(* PLC project DBISFactory.project, CODESYS CODESYS V3.5 SP10 Patch 5 *)
(* stored: creationDateTime 2019-03-07T13:49:44.3534286, modificationDateTime 2019-03-07T13:47:37.4051931 *)

(* values of BatchJobState: NULL: NULL always expresses that the object has not been initialized yet; WAITING: BatchJob has been initialized and is waiting to be executed; STARTED: BatchJob has been started and is being executed now; PAUSED: BatchJob has been paused during execution; ABORTED: BatchJob has been aborted. This may happen at any time; FINISHED: BatchJob has been finished *)

(* States of a BatchJob Copyright (c) 2019 Manuel Goester, Michael Witt, Klaus Kammerer Institute of Databases and Information Systems, Ulm University, Germany Permission is hereby granted, free of charge, to any person obtaining a copy of this software and associated documentation files (the "Software"), to deal in the Software without restriction, including without limitation the rights to use, copy, modify, merge, publish, distribute, sublicense, and/or sell copies of the Software, and to permit persons to whom the Software is furnished to do so, subject to the following conditions: The above copyright notice and this permission notice shall be included in all copies or substantial portions of the Software. THE SOFTWARE IS PROVIDED "AS IS", WITHOUT WARRANTY OF ANY KIND, EXPRESS OR IMPLIED, INCLUDING BUT NOT LIMITED TO THE WARRANTIES OF MERCHANTABILITY, FITNESS FOR A PARTICULAR PURPOSE AND NONINFRINGEMENT. IN NO EVENT SHALL THE AUTHORS OR COPYRIGHT HOLDERS BE LIABLE FOR ANY CLAIM, DAMAGES OR OTHER LIABILITY, WHETHER IN AN ACTION OF CONTRACT, TORT OR OTHERWISE, ARISING FROM, OUT OF OR IN CONNECTION WITH THE SOFTWARE OR THE USE OR OTHER DEALINGS IN THE SOFTWARE. *)
TYPE BatchJobState : (NULL := 0, WAITING := 1, STARTED := 2, PAUSED := 3, ABORTED := 4, FINISHED := 5);
END_TYPE

(* Execution modes of a BatchJob Copyright (c) 2019 Manuel Goester, Michael Witt, Klaus Kammerer Institute of Databases and Information Systems, Ulm University, Germany Permission is hereby granted, free of charge, to any person obtaining a copy of this software and associated documentation files (the "Software"), to deal in the Software without restriction, including without limitation the rights to use, copy, modify, merge, publish, distribute, sublicense, and/or sell copies of the Software, and to permit persons to whom the Software is furnished to do so, subject to the following conditions: The above copyright notice and this permission notice shall be included in all copies or substantial portions of the Software. THE SOFTWARE IS PROVIDED "AS IS", WITHOUT WARRANTY OF ANY KIND, EXPRESS OR IMPLIED, INCLUDING BUT NOT LIMITED TO THE WARRANTIES OF MERCHANTABILITY, FITNESS FOR A PARTICULAR PURPOSE AND NONINFRINGEMENT. IN NO EVENT SHALL THE AUTHORS OR COPYRIGHT HOLDERS BE LIABLE FOR ANY CLAIM, DAMAGES OR OTHER LIABILITY, WHETHER IN AN ACTION OF CONTRACT, TORT OR OTHERWISE, ARISING FROM, OUT OF OR IN CONNECTION WITH THE SOFTWARE OR THE USE OR OTHER DEALINGS IN THE SOFTWARE. *)
TYPE ExecutionMode : (single := 0, multi := 1, sorting := 2);
END_TYPE

(* A Format defines the execution options of a workpiece Copyright (c) 2019 Manuel Goester, Michael Witt, Klaus Kammerer Institute of Databases and Information Systems, Ulm University, Germany Permission is hereby granted, free of charge, to any person obtaining a copy of this software and associated documentation files (the "Software"), to deal in the Software without restriction, including without limitation the rights to use, copy, modify, merge, publish, distribute, sublicense, and/or sell copies of the Software, and to permit persons to whom the Software is furnished to do so, subject to the following conditions: The above copyright notice and this permission notice shall be included in all copies or substantial portions of the Software. THE SOFTWARE IS PROVIDED "AS IS", WITHOUT WARRANTY OF ANY KIND, EXPRESS OR IMPLIED, INCLUDING BUT NOT LIMITED TO THE WARRANTIES OF MERCHANTABILITY, FITNESS FOR A PARTICULAR PURPOSE AND NONINFRINGEMENT. IN NO EVENT SHALL THE AUTHORS OR COPYRIGHT HOLDERS BE LIABLE FOR ANY CLAIM, DAMAGES OR OTHER LIABILITY, WHETHER IN AN ACTION OF CONTRACT, TORT OR OTHERWISE, ARISING FROM, OUT OF OR IN CONNECTION WITH THE SOFTWARE OR THE USE OR OTHER DEALINGS IN THE SOFTWARE. *)
TYPE Format : STRUCT
  furEnabled : BOOL;
  sawEnabled : BOOL;
  colorCheckEnabled : BOOL;
  ejectEnabled : BOOL;
  furDuration : TIME;
  sawDuration : TIME;
END_STRUCT;
END_TYPE

(* Configured BatchJobs are stored in a BatchJobQueue Copyright (c) 2019 Manuel Goester, Michael Witt, Klaus Kammerer Institute of Databases and Information Systems, Ulm University, Germany Permission is hereby granted, free of charge, to any person obtaining a copy of this software and associated documentation files (the "Software"), to deal in the Software without restriction, including without limitation the rights to use, copy, modify, merge, publish, distribute, sublicense, and/or sell copies of the Software, and to permit persons to whom the Software is furnished to do so, subject to the following conditions: The above copyright notice and this permission notice shall be included in all copies or substantial portions of the Software. THE SOFTWARE IS PROVIDED "AS IS", WITHOUT WARRANTY OF ANY KIND, EXPRESS OR IMPLIED, INCLUDING BUT NOT LIMITED TO THE WARRANTIES OF MERCHANTABILITY, FITNESS FOR A PARTICULAR PURPOSE AND NONINFRINGEMENT. IN NO EVENT SHALL THE AUTHORS OR COPYRIGHT HOLDERS BE LIABLE FOR ANY CLAIM, DAMAGES OR OTHER LIABILITY, WHETHER IN AN ACTION OF CONTRACT, TORT OR OTHERWISE, ARISING FROM, OUT OF OR IN CONNECTION WITH THE SOFTWARE OR THE USE OR OTHER DEALINGS IN THE SOFTWARE. *)
TYPE BatchJobQueue : STRUCT
  batchJobs : ARRAY[1..512] OF BatchJob;  (* batch job queue *)
  nextFreePos : INT := 1;  (* next free place in batchJobs *)
  amountBatchJobs : INT := 0;  (* amount of batch jobs currently being in queue *)
  full : BOOL;  (* true if batchJobs array full *)
END_STRUCT;
END_TYPE

(* Datastructure describing the "real world workpiece" Copyright (c) 2019 Manuel Goester, Michael Witt, Klaus Kammerer Institute of Databases and Information Systems, Ulm University, Germany Permission is hereby granted, free of charge, to any person obtaining a copy of this software and associated documentation files (the "Software"), to deal in the Software without restriction, including without limitation the rights to use, copy, modify, merge, publish, distribute, sublicense, and/or sell copies of the Software, and to permit persons to whom the Software is furnished to do so, subject to the following conditions: The above copyright notice and this permission notice shall be included in all copies or substantial portions of the Software. THE SOFTWARE IS PROVIDED "AS IS", WITHOUT WARRANTY OF ANY KIND, EXPRESS OR IMPLIED, INCLUDING BUT NOT LIMITED TO THE WARRANTIES OF MERCHANTABILITY, FITNESS FOR A PARTICULAR PURPOSE AND NONINFRINGEMENT. IN NO EVENT SHALL THE AUTHORS OR COPYRIGHT HOLDERS BE LIABLE FOR ANY CLAIM, DAMAGES OR OTHER LIABILITY, WHETHER IN AN ACTION OF CONTRACT, TORT OR OTHERWISE, ARISING FROM, OUT OF OR IN CONNECTION WITH THE SOFTWARE OR THE USE OR OTHER DEALINGS IN THE SOFTWARE. *)
TYPE Workpiece : STRUCT
  color : STRING(7);  (* red, blue, white or unknown *)
  linePos : INT;  (* 0 = high rack, 1 = vacuum gripper, 2 = Furnace, 3 = sorting line *)
  sortingLinePos : INT;  (* position in high rack at begin and end of batch job (1,1) (1,2) (1,3) (2,1) (2,2) (2,3) (3,1) (3,2) (3,3) highRackPos: ARRAY [1..2] OF INT; highRackPosEnd: ARRAY [1..2] OF INT; position in sorting line *)
  state : W_State;
  startPos : RackPos;
  endPos : RackPos;
  format : Format;  (* defines which actions will be executed and how long *)
END_STRUCT;
END_TYPE

(* A BatchJob is a task which shall be executed on the production lane. It consists of a set of workpieces, which are executed by the production lane in a certain mode. Copyright (c) 2019 Manuel Goester, Michael Witt, Klaus Kammerer Institute of Databases and Information Systems, Ulm University, Germany Permission is hereby granted, free of charge, to any person obtaining a copy of this software and associated documentation files (the "Software"), to deal in the Software without restriction, including without limitation the rights to use, copy, modify, merge, publish, distribute, sublicense, and/or sell copies of the Software, and to permit persons to whom the Software is furnished to do so, subject to the following conditions: The above copyright notice and this permission notice shall be included in all copies or substantial portions of the Software. THE SOFTWARE IS PROVIDED "AS IS", WITHOUT WARRANTY OF ANY KIND, EXPRESS OR IMPLIED, INCLUDING BUT NOT LIMITED TO THE WARRANTIES OF MERCHANTABILITY, FITNESS FOR A PARTICULAR PURPOSE AND NONINFRINGEMENT. IN NO EVENT SHALL THE AUTHORS OR COPYRIGHT HOLDERS BE LIABLE FOR ANY CLAIM, DAMAGES OR OTHER LIABILITY, WHETHER IN AN ACTION OF CONTRACT, TORT OR OTHERWISE, ARISING FROM, OUT OF OR IN CONNECTION WITH THE SOFTWARE OR THE USE OR OTHER DEALINGS IN THE SOFTWARE. *)
TYPE BatchJob : STRUCT
  batchSize : INT;  (* amount of workpieces in batch job *)
  workpieces : ARRAY[1..9] OF Workpiece;  (* workpieces being processed *)
  nextFreeWPos : INT := 1;  (* next free place in workpieces *)
  nextNotProcessedIdx : INT := 1;  (* index in workpieces of the next workpiece whose production has not started yet *)
  amountFinishedW : INT := 0;  (* states how many workpieces are already finished *)
  mode : ExecutionMode := ExecutionMode.single;  (* type of execution *)
  timeCreated : DT;  (* time when created *)
  timeStarted : DT;  (* time when started *)
  timeFinished : DT;  (* time when finished / aborted *)
  pauseDuration : TIME;  (* states the time how long the batch job was in pause state *)
  duration : TIME;  (* states how long the batch job took *)
  state : BatchJobState := BatchJobState.NULL;  (* state of batch job *)
END_STRUCT;
END_TYPE

(* values of RackPos: UP: there are different values for up position or down position at rack or at conveyor see: HR_FBs/HR_MOVE_TO_POS *)

(* Positions in high rack. Used for HR navigation Copyright (c) 2019 Manuel Goester, Michael Witt, Klaus Kammerer Institute of Databases and Information Systems, Ulm University, Germany Permission is hereby granted, free of charge, to any person obtaining a copy of this software and associated documentation files (the "Software"), to deal in the Software without restriction, including without limitation the rights to use, copy, modify, merge, publish, distribute, sublicense, and/or sell copies of the Software, and to permit persons to whom the Software is furnished to do so, subject to the following conditions: The above copyright notice and this permission notice shall be included in all copies or substantial portions of the Software. THE SOFTWARE IS PROVIDED "AS IS", WITHOUT WARRANTY OF ANY KIND, EXPRESS OR IMPLIED, INCLUDING BUT NOT LIMITED TO THE WARRANTIES OF MERCHANTABILITY, FITNESS FOR A PARTICULAR PURPOSE AND NONINFRINGEMENT. IN NO EVENT SHALL THE AUTHORS OR COPYRIGHT HOLDERS BE LIABLE FOR ANY CLAIM, DAMAGES OR OTHER LIABILITY, WHETHER IN AN ACTION OF CONTRACT, TORT OR OTHERWISE, ARISING FROM, OUT OF OR IN CONNECTION WITH THE SOFTWARE OR THE USE OR OTHER DEALINGS IN THE SOFTWARE. *)
TYPE RackPos : (NULL := 0, RACK_11 := 1, RACK_12 := 2, RACK_13 := 3, RACK_21 := 4, RACK_22 := 5, RACK_23 := 6, RACK_31 := 7, RACK_32 := 8, RACK_33 := 9, CONVEYOR := 10, UP := 11, DOWN := 12);
END_TYPE

(* values of HR_State: NULL: NULL always expresses that the Object has not been initialized yet; AT_DEFAULT_POS: used in single mode; WAIT_FOR_VG_TO_BRING_W: used in multi mode; GET_W: <-- also used in single mode; FINISHED_SORTING_MODE: used in sorting mode *)

(* States of the HR (High Rack) station. Copyright (c) 2019 Manuel Goester, Michael Witt, Klaus Kammerer Institute of Databases and Information Systems, Ulm University, Germany Permission is hereby granted, free of charge, to any person obtaining a copy of this software and associated documentation files (the "Software"), to deal in the Software without restriction, including without limitation the rights to use, copy, modify, merge, publish, distribute, sublicense, and/or sell copies of the Software, and to permit persons to whom the Software is furnished to do so, subject to the following conditions: The above copyright notice and this permission notice shall be included in all copies or substantial portions of the Software. THE SOFTWARE IS PROVIDED "AS IS", WITHOUT WARRANTY OF ANY KIND, EXPRESS OR IMPLIED, INCLUDING BUT NOT LIMITED TO THE WARRANTIES OF MERCHANTABILITY, FITNESS FOR A PARTICULAR PURPOSE AND NONINFRINGEMENT. IN NO EVENT SHALL THE AUTHORS OR COPYRIGHT HOLDERS BE LIABLE FOR ANY CLAIM, DAMAGES OR OTHER LIABILITY, WHETHER IN AN ACTION OF CONTRACT, TORT OR OTHERWISE, ARISING FROM, OUT OF OR IN CONNECTION WITH THE SOFTWARE OR THE USE OR OTHER DEALINGS IN THE SOFTWARE. *)
TYPE HR_State : (NULL := 0, AT_DEFAULT_POS := 1, FINISHED_SINGLE_MODE := 2, AT_CONVEYOR_BOX_FULL := 25, AT_CONVEYOR_BOX_EMPTY := 26, WAIT_FOR_VG_TO_BRING_W := 8, GET_W := 9, GET_BOX := 10, STORE_W := 20, STORE_BOX := 19, WAIT_FOR_VG_TO_PICK_UP_W := 11, READY := 12, FINISHED_SORTING_MODE := 40, SORTING := 41);
END_TYPE

(* values of VG_State: NULL: NULL always expresses that the object has not been initialized yet; FROM_HR_TO_EJECT: used in single mode; TO_FUR_PUT_W: used in multi mode; READY: ready if VG is at default pos or if VG put down a workpiece at HR --> VG is ready for next workpiece; AT_DEFAULT_POS: used in single and multi mode *)

(* States of the VG (Vacuum Gripper) station. Copyright (c) 2019 Manuel Goester, Michael Witt, Klaus Kammerer Institute of Databases and Information Systems, Ulm University, Germany Permission is hereby granted, free of charge, to any person obtaining a copy of this software and associated documentation files (the "Software"), to deal in the Software without restriction, including without limitation the rights to use, copy, modify, merge, publish, distribute, sublicense, and/or sell copies of the Software, and to permit persons to whom the Software is furnished to do so, subject to the following conditions: The above copyright notice and this permission notice shall be included in all copies or substantial portions of the Software. THE SOFTWARE IS PROVIDED "AS IS", WITHOUT WARRANTY OF ANY KIND, EXPRESS OR IMPLIED, INCLUDING BUT NOT LIMITED TO THE WARRANTIES OF MERCHANTABILITY, FITNESS FOR A PARTICULAR PURPOSE AND NONINFRINGEMENT. IN NO EVENT SHALL THE AUTHORS OR COPYRIGHT HOLDERS BE LIABLE FOR ANY CLAIM, DAMAGES OR OTHER LIABILITY, WHETHER IN AN ACTION OF CONTRACT, TORT OR OTHERWISE, ARISING FROM, OUT OF OR IN CONNECTION WITH THE SOFTWARE OR THE USE OR OTHER DEALINGS IN THE SOFTWARE. *)
TYPE VG_State : (NULL := 0, FROM_HR_TO_EJECT := 6, AT_HR := 30, FROM_HR_TO_FUR := 31, AT_SL_OUTPUT_1 := 32, AT_SL_OUTPUT_2 := 33, AT_SL_OUTPUT_3 := 34, WAIT_FOR_SL := 35, AT_EJECT_1 := 36, AT_EJECT_2 := 37, AT_EJECT_3 := 38, TO_SL_OUTPUT_1 := 39, TO_SL_OUTPUT_2 := 40, TO_SL_OUTPUT_3 := 41, FROM_DEFAULT_POS_TO_HR := 43, GET_W_FROM_HR := 44, ABOVE_SL := 56, FROM_SL_TO_HR := 57, DROPPING_W_TO_HR := 59, TO_FUR_PUT_W := 8, TO_FUR_PUT_W_FINISHED := 9, TO_SL_TAKE_W := 10, TO_SL_TAKE_W_FINISHED := 11, TO_HR_PUT_W := 12, TO_HR_PUT_W_FINISHED := 13, TO_HR_TAKE_W := 14, TO_HR_TAKE_W_FINISHED := 15, TO_EJECT := 16, TO_EJECT_FINISHED := 17, TO_SL := 45, READY := 18, AT_DEFAULT_POS := 1, TO_DEFAULT_POS := 5);
END_TYPE

(* values of FUR_State: NULL: TODO : Use these states also in multi mode NULL always expresses that the Object has not been initialized yet; FUR_WAITING_FOR_W: used in single mode FUR is ready to take a new workpiece; FUR_LB_PASSED: Workpiece passed the lightbarrier at waggon; FUR_WAGON_INSIDE: used in single and multi mode Wagon is inside of burner; FUR_BURNED: Furnace is finished with buring the workpiece; FUR_WAGON_OUTSIDE: Wagon is outside of burner; FUR_SUCCER_AT_FUR: used in single mode furnace succer is at furnace; FUR_SUCCER_DOWN_AT_FUR: furnace succer picks up workpiece; FUR_SUCCER_TO_ROTARY_DESK: furnace succer on the way to rotary desk; FUR_SUCCER_AT_ROTARY_DESK: furnace succer at rotary desk; FUR_SUCCER_DOWN_AT_RD: furnace succer puts down workpiece; FUR_SAW_FINISHED: saw has been finished; FUR_SKIP_SAW: saw has been skipped; FUR_W_FINISHED_BACK_TO_DEFAULT: station has finished processing this workpiece *)

(* States of the FUR (Furnace) station. The station is composed of a burner, succer, rotary desk and saw. Copyright (c) 2019 Manuel Goester, Michael Witt, Klaus Kammerer Institute of Databases and Information Systems, Ulm University, Germany Permission is hereby granted, free of charge, to any person obtaining a copy of this software and associated documentation files (the "Software"), to deal in the Software without restriction, including without limitation the rights to use, copy, modify, merge, publish, distribute, sublicense, and/or sell copies of the Software, and to permit persons to whom the Software is furnished to do so, subject to the following conditions: The above copyright notice and this permission notice shall be included in all copies or substantial portions of the Software. THE SOFTWARE IS PROVIDED "AS IS", WITHOUT WARRANTY OF ANY KIND, EXPRESS OR IMPLIED, INCLUDING BUT NOT LIMITED TO THE WARRANTIES OF MERCHANTABILITY, FITNESS FOR A PARTICULAR PURPOSE AND NONINFRINGEMENT. IN NO EVENT SHALL THE AUTHORS OR COPYRIGHT HOLDERS BE LIABLE FOR ANY CLAIM, DAMAGES OR OTHER LIABILITY, WHETHER IN AN ACTION OF CONTRACT, TORT OR OTHERWISE, ARISING FROM, OUT OF OR IN CONNECTION WITH THE SOFTWARE OR THE USE OR OTHER DEALINGS IN THE SOFTWARE. *)
TYPE FUR_State : (NULL := 0, FUR_WAITING_FOR_W := 1, FUR_LB_PASSED := 2, FUR_WAGON_INSIDE := 3, FUR_BURNED := 4, FUR_WAGON_OUTSIDE := 5, FUR_SUCCER_AT_FUR := 6, FUR_SUCCER_DOWN_AT_FUR := 7, FUR_SUCCER_UP_AT_FUR := 8, FUR_SUCCER_TO_ROTARY_DESK := 9, FUR_SUCCER_AT_ROTARY_DESK := 10, FUR_SUCCER_DOWN_AT_RD := 11, FUR_SUCCER_UP_AT_RD := 12, FUR_SAW_FINISHED := 13, FUR_SKIP_SAW := 14, FUR_W_FINISHED_BACK_TO_DEFAULT := 15);
END_TYPE

(* values of SL_State: NULL: NULL always expresses that the object has not been initialized yet; WAITING_FOR_W: SL is ready to process a new workpiece; W_AT_LB: Lightbarrier at SL entry has been passed by a workpiece; THROW_OUT: if no color was detected, the workpiece will be thrown out to trash; W_RECEIVED: SL got a workpiece to process it *)

(* States of the SL (Sorting Line) station. Copyright (c) 2019 Manuel Goester, Michael Witt, Klaus Kammerer Institute of Databases and Information Systems, Ulm University, Germany Permission is hereby granted, free of charge, to any person obtaining a copy of this software and associated documentation files (the "Software"), to deal in the Software without restriction, including without limitation the rights to use, copy, modify, merge, publish, distribute, sublicense, and/or sell copies of the Software, and to permit persons to whom the Software is furnished to do so, subject to the following conditions: The above copyright notice and this permission notice shall be included in all copies or substantial portions of the Software. THE SOFTWARE IS PROVIDED "AS IS", WITHOUT WARRANTY OF ANY KIND, EXPRESS OR IMPLIED, INCLUDING BUT NOT LIMITED TO THE WARRANTIES OF MERCHANTABILITY, FITNESS FOR A PARTICULAR PURPOSE AND NONINFRINGEMENT. IN NO EVENT SHALL THE AUTHORS OR COPYRIGHT HOLDERS BE LIABLE FOR ANY CLAIM, DAMAGES OR OTHER LIABILITY, WHETHER IN AN ACTION OF CONTRACT, TORT OR OTHERWISE, ARISING FROM, OUT OF OR IN CONNECTION WITH THE SOFTWARE OR THE USE OR OTHER DEALINGS IN THE SOFTWARE. *)
TYPE SL_State : (NULL := 0, WAITING_FOR_W := 1, W_AT_LB := 2, W_AT_COLORCHECK := 3, COLORCHECK_FINISHED := 4, W_READY_FOR_SORTING := 5, THROW_OUT := 6, SORTING := 7, WAITING_FOR_VG_TO_PICK_UP_W := 8, EJECT := 9, EJECTED := 10, W_RECEIVED := 11);
END_TYPE

(* values of W_State: NULL: NULL always expresses that the object has not been initialized yet; AT_RACK_11: states at HR; FROM_RACK_TO_CONVEYOR: NOT used; AT_HR: states at VG NOT used; AT_FUR_IN_WAGON: states at FUR; AT_SL_AT_ENTRY_LIGHT_BARRIER: states at SL not used; AT_EJECT_1: states at EJECT point not used *)

(* Workpiece States Copyright (c) 2019 Manuel Goester, Michael Witt, Klaus Kammerer Institute of Databases and Information Systems, Ulm University, Germany Permission is hereby granted, free of charge, to any person obtaining a copy of this software and associated documentation files (the "Software"), to deal in the Software without restriction, including without limitation the rights to use, copy, modify, merge, publish, distribute, sublicense, and/or sell copies of the Software, and to permit persons to whom the Software is furnished to do so, subject to the following conditions: The above copyright notice and this permission notice shall be included in all copies or substantial portions of the Software. THE SOFTWARE IS PROVIDED "AS IS", WITHOUT WARRANTY OF ANY KIND, EXPRESS OR IMPLIED, INCLUDING BUT NOT LIMITED TO THE WARRANTIES OF MERCHANTABILITY, FITNESS FOR A PARTICULAR PURPOSE AND NONINFRINGEMENT. IN NO EVENT SHALL THE AUTHORS OR COPYRIGHT HOLDERS BE LIABLE FOR ANY CLAIM, DAMAGES OR OTHER LIABILITY, WHETHER IN AN ACTION OF CONTRACT, TORT OR OTHERWISE, ARISING FROM, OUT OF OR IN CONNECTION WITH THE SOFTWARE OR THE USE OR OTHER DEALINGS IN THE SOFTWARE. *)
TYPE W_State : (NULL := 0, AT_RACK_11 := 111, AT_RACK_12 := 112, AT_RACK_13 := 113, AT_RACK_21 := 121, AT_RACK_22 := 122, AT_RACK_23 := 123, AT_RACK_31 := 131, AT_RACK_32 := 132, AT_RACK_33 := 133, FROM_RACK_TO_CONVEYOR := 140, AT_CONVEYOR_INSIDE := 141, FROM_CONVEYOR_INSIDE_TO_OUTSIDE := 142, AT_CONVEYOR_OUTSIDE := 143, FROM_CONVEYOR_OUTSIDE_TO_INSIDE := 144, AT_HR := 200, FROM_HR_TO_FUR := 201, FROM_SL_OUTPUT_TO_HR := 202, FROM_SL_OUTPUT_1_TO_HR := 203, FROM_SL_OUTPUT_2_TO_HR := 204, FROM_SL_OUTPUT_3_TO_HR := 205, FROM_SL_TO_EJECT := 206, FROM_SL_OUTPUT_1_TO_EJECT := 207, FROM_SL_OUTPUT_2_TO_EJECT := 208, FROM_SL_OUTPUT_3_TO_EJECT := 209, FROM_FUR_TO_HR := 210, AT_FUR_IN_WAGON := 300, AT_FUR_IN_FUR := 301, AT_FUR_ATTACHED_TO_SUCCER := 302, AT_FUR_ON_ROTARY_DESK := 303, AT_FUR_AT_SAW := 304, AT_FUR_ON_CONVEYOR := 305, AT_SL_AT_ENTRY_LIGHT_BARRIER := 400, AT_SL_AT_COLORCHECK := 401, AT_SL_AT_EXIT_LIGHT_BARRIER := 402, AT_SL_OUTPUT_1 := 403, AT_SL_OUTPUT_2 := 404, AT_SL_OUTPUT_3 := 405, AT_SL_OUTPUT_TRASH := 406, AT_EJECT_1 := 500, AT_EJECT_2 := 501, AT_EJECT_3 := 502);
END_TYPE

(* values of TC_State: NULL: NULL always expresses that the Object has not been initialized yet; W_LOADED: TC has loaded a new workpiece to HR; WAIT_UNTIL_W_FINISHED: TC is waiting until the workpiece has been processed; LOAD_NEXT_W: TC is loading a new workpiece *)

(* States of TC (Task Configurator). Copyright (c) 2019 Manuel Goester, Michael Witt, Klaus Kammerer Institute of Databases and Information Systems, Ulm University, Germany Permission is hereby granted, free of charge, to any person obtaining a copy of this software and associated documentation files (the "Software"), to deal in the Software without restriction, including without limitation the rights to use, copy, modify, merge, publish, distribute, sublicense, and/or sell copies of the Software, and to permit persons to whom the Software is furnished to do so, subject to the following conditions: The above copyright notice and this permission notice shall be included in all copies or substantial portions of the Software. THE SOFTWARE IS PROVIDED "AS IS", WITHOUT WARRANTY OF ANY KIND, EXPRESS OR IMPLIED, INCLUDING BUT NOT LIMITED TO THE WARRANTIES OF MERCHANTABILITY, FITNESS FOR A PARTICULAR PURPOSE AND NONINFRINGEMENT. IN NO EVENT SHALL THE AUTHORS OR COPYRIGHT HOLDERS BE LIABLE FOR ANY CLAIM, DAMAGES OR OTHER LIABILITY, WHETHER IN AN ACTION OF CONTRACT, TORT OR OTHERWISE, ARISING FROM, OUT OF OR IN CONNECTION WITH THE SOFTWARE OR THE USE OR OTHER DEALINGS IN THE SOFTWARE. *)
TYPE TC_State : (NULL := 0, W_LOADED := 1, WAIT_UNTIL_W_FINISHED := 2, LOAD_NEXT_W := 3);
END_TYPE

PROGRAM FUR_SINGLE_MODE
  VAR
    trigger : INT;
    timer : TON;
    sawStopped : BOOL;
    wAtSL : BOOL;
    fin : BOOL;
  END_VAR

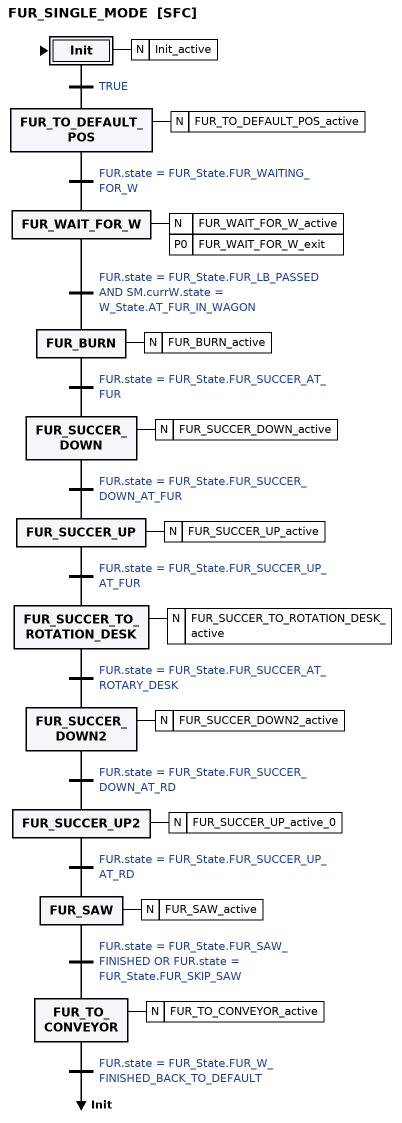
INITIAL_STEP Init:
  Init_active(N);
END_STEP
TRANSITION FROM Init TO FUR_TO_DEFAULT_POS
  := TRUE;
END_TRANSITION
STEP FUR_TO_DEFAULT_POS:
  FUR_TO_DEFAULT_POS_active(N);
END_STEP
TRANSITION FROM FUR_TO_DEFAULT_POS TO FUR_WAIT_FOR_W
  := FUR.state = FUR_State.FUR_WAITING_FOR_W;
END_TRANSITION
STEP FUR_WAIT_FOR_W:
  FUR_WAIT_FOR_W_active(N);
  FUR_WAIT_FOR_W_exit(P0);
END_STEP
TRANSITION FROM FUR_WAIT_FOR_W TO FUR_BURN
  := FUR.state = FUR_State.FUR_LB_PASSED AND SM.currW.state = W_State.AT_FUR_IN_WAGON;
END_TRANSITION
STEP FUR_BURN:
  FUR_BURN_active(N);
END_STEP
TRANSITION FROM FUR_BURN TO FUR_SUCCER_DOWN
  := FUR.state = FUR_State.FUR_SUCCER_AT_FUR;
END_TRANSITION
STEP FUR_SUCCER_DOWN:
  FUR_SUCCER_DOWN_active(N);
END_STEP
TRANSITION FROM FUR_SUCCER_DOWN TO FUR_SUCCER_UP
  := FUR.state = FUR_State.FUR_SUCCER_DOWN_AT_FUR;
END_TRANSITION
STEP FUR_SUCCER_UP:
  FUR_SUCCER_UP_active(N);
END_STEP
TRANSITION FROM FUR_SUCCER_UP TO FUR_SUCCER_TO_ROTATION_DESK
  := FUR.state = FUR_State.FUR_SUCCER_UP_AT_FUR;
END_TRANSITION
STEP FUR_SUCCER_TO_ROTATION_DESK:
  FUR_SUCCER_TO_ROTATION_DESK_active(N);
END_STEP
TRANSITION FROM FUR_SUCCER_TO_ROTATION_DESK TO FUR_SUCCER_DOWN2
  := FUR.state = FUR_State.FUR_SUCCER_AT_ROTARY_DESK;
END_TRANSITION
STEP FUR_SUCCER_DOWN2:
  FUR_SUCCER_DOWN2_active(N);
END_STEP
TRANSITION FROM FUR_SUCCER_DOWN2 TO FUR_SUCCER_UP2
  := FUR.state = FUR_State.FUR_SUCCER_DOWN_AT_RD;
END_TRANSITION
STEP FUR_SUCCER_UP2:
  FUR_SUCCER_UP_active_0(N);
END_STEP
TRANSITION FROM FUR_SUCCER_UP2 TO FUR_SAW
  := FUR.state = FUR_State.FUR_SUCCER_UP_AT_RD;
END_TRANSITION
STEP FUR_SAW:
  FUR_SAW_active(N);
END_STEP
TRANSITION FROM FUR_SAW TO FUR_TO_CONVEYOR
  := FUR.state = FUR_State.FUR_SAW_FINISHED OR FUR.state = FUR_State.FUR_SKIP_SAW;
END_TRANSITION
STEP FUR_TO_CONVEYOR:
  FUR_TO_CONVEYOR_active(N);
END_STEP
TRANSITION FROM FUR_TO_CONVEYOR TO Init
  := FUR.state = FUR_State.FUR_W_FINISHED_BACK_TO_DEFAULT;
END_TRANSITION

ACTION FUR_SUCCER_UP_active_0:
                      (*
Copyright (c) 2019 Manuel Goester, Michael Witt, Klaus Kammerer
Institute of Databases and Information Systems, Ulm University, Germany

Permission is hereby granted, free of charge, to any person obtaining a copy 
of this software and associated documentation files (the "Software"), to deal 
in the Software without restriction, including without limitation the rights 
to use, copy, modify, merge, publish, distribute, sublicense, and/or sell 
copies of the Software, and to permit persons to whom the Software is 
furnished to do so, subject to the following conditions:

The above copyright notice and this permission notice shall be included in 
all copies or substantial portions of the Software.

THE SOFTWARE IS PROVIDED "AS IS", WITHOUT WARRANTY OF ANY KIND, EXPRESS OR 
IMPLIED, INCLUDING BUT NOT LIMITED TO THE WARRANTIES OF MERCHANTABILITY, 
FITNESS FOR A PARTICULAR PURPOSE AND NONINFRINGEMENT. IN NO EVENT SHALL THE 
AUTHORS OR COPYRIGHT HOLDERS BE LIABLE FOR ANY CLAIM, DAMAGES OR OTHER 
LIABILITY, WHETHER IN AN ACTION OF CONTRACT, TORT OR OTHERWISE, ARISING FROM, 
OUT OF OR IN CONNECTION WITH THE SOFTWARE OR THE USE OR OTHER DEALINGS 
IN THE SOFTWARE.
*)
timer(IN:= TRUE, PT := T#200MS);
IF NOT(timer.Q = FALSE AND timer.IN) THEN
	timer(IN:= FALSE);
	FUR.state := FUR_State.FUR_SUCCER_UP_AT_RD;
	SM.currW.state := W_State.AT_FUR_ON_ROTARY_DESK;
END_IF

                    
END_ACTION

ACTION FUR_SUCCER_TO_ROTATION_DESK_active:
                      (*
Copyright (c) 2019 Manuel Goester, Michael Witt, Klaus Kammerer
Institute of Databases and Information Systems, Ulm University, Germany

Permission is hereby granted, free of charge, to any person obtaining a copy 
of this software and associated documentation files (the "Software"), to deal 
in the Software without restriction, including without limitation the rights 
to use, copy, modify, merge, publish, distribute, sublicense, and/or sell 
copies of the Software, and to permit persons to whom the Software is 
furnished to do so, subject to the following conditions:

The above copyright notice and this permission notice shall be included in 
all copies or substantial portions of the Software.

THE SOFTWARE IS PROVIDED "AS IS", WITHOUT WARRANTY OF ANY KIND, EXPRESS OR 
IMPLIED, INCLUDING BUT NOT LIMITED TO THE WARRANTIES OF MERCHANTABILITY, 
FITNESS FOR A PARTICULAR PURPOSE AND NONINFRINGEMENT. IN NO EVENT SHALL THE 
AUTHORS OR COPYRIGHT HOLDERS BE LIABLE FOR ANY CLAIM, DAMAGES OR OTHER 
LIABILITY, WHETHER IN AN ACTION OF CONTRACT, TORT OR OTHERWISE, ARISING FROM, 
OUT OF OR IN CONNECTION WITH THE SOFTWARE OR THE USE OR OTHER DEALINGS 
IN THE SOFTWARE.
*)
IF  NOT(FUR.sSuckerPosRa) THEN
	FUR.mSuckertoRa := TRUE;
	FUR.state := FUR_State.FUR_SUCCER_TO_ROTARY_DESK;
ELSE
	FUR.mSuckertoRa := FALSE;
	FUR.compressor := FALSE;
	FUR.valveLowering := TRUE;
	FUR.state := FUR_State.FUR_SUCCER_AT_ROTARY_DESK;
END_IF
                    
END_ACTION

ACTION FUR_SAW_active:
                      (*
Copyright (c) 2019 Manuel Goester, Michael Witt, Klaus Kammerer
Institute of Databases and Information Systems, Ulm University, Germany

Permission is hereby granted, free of charge, to any person obtaining a copy 
of this software and associated documentation files (the "Software"), to deal 
in the Software without restriction, including without limitation the rights 
to use, copy, modify, merge, publish, distribute, sublicense, and/or sell 
copies of the Software, and to permit persons to whom the Software is 
furnished to do so, subject to the following conditions:

The above copyright notice and this permission notice shall be included in 
all copies or substantial portions of the Software.

THE SOFTWARE IS PROVIDED "AS IS", WITHOUT WARRANTY OF ANY KIND, EXPRESS OR 
IMPLIED, INCLUDING BUT NOT LIMITED TO THE WARRANTIES OF MERCHANTABILITY, 
FITNESS FOR A PARTICULAR PURPOSE AND NONINFRINGEMENT. IN NO EVENT SHALL THE 
AUTHORS OR COPYRIGHT HOLDERS BE LIABLE FOR ANY CLAIM, DAMAGES OR OTHER 
LIABILITY, WHETHER IN AN ACTION OF CONTRACT, TORT OR OTHERWISE, ARISING FROM, 
OUT OF OR IN CONNECTION WITH THE SOFTWARE OR THE USE OR OTHER DEALINGS 
IN THE SOFTWARE.
*)
IF SM.currW.format.sawEnabled THEN
	SM.currW.state := W_State.AT_FUR_AT_SAW;
	IF NOT(FUR.sRaPosSaw) THEN
		FUR.mRaClockwise := TRUE;
	ELSE
		FUR.mRaClockwise := FALSE;
		sawStopped := TRUE;
	END_IF
	
	IF sawStopped THEN
		timer(IN:= TRUE, PT := SM.currW.format.sawDuration);
		FUR.mSaw := TRUE;
		
		IF NOT(timer.Q = FALSE AND timer.IN) THEN
			timer(IN:=FALSE);
			FUR.mSaw := FALSE;
			sawStopped := FALSE;
			FUR.state := FUR_State.FUR_SAW_FINISHED;
		END_IF
	END_IF
ELSE
	// skip saw
	FUR.state := FUR_State.FUR_SKIP_SAW;
END_IF

                    
END_ACTION

ACTION FUR_WAIT_FOR_W_exit:
                      (*
Copyright (c) 2019 Manuel Goester, Michael Witt, Klaus Kammerer
Institute of Databases and Information Systems, Ulm University, Germany

Permission is hereby granted, free of charge, to any person obtaining a copy 
of this software and associated documentation files (the "Software"), to deal 
in the Software without restriction, including without limitation the rights 
to use, copy, modify, merge, publish, distribute, sublicense, and/or sell 
copies of the Software, and to permit persons to whom the Software is 
furnished to do so, subject to the following conditions:

The above copyright notice and this permission notice shall be included in 
all copies or substantial portions of the Software.

THE SOFTWARE IS PROVIDED "AS IS", WITHOUT WARRANTY OF ANY KIND, EXPRESS OR 
IMPLIED, INCLUDING BUT NOT LIMITED TO THE WARRANTIES OF MERCHANTABILITY, 
FITNESS FOR A PARTICULAR PURPOSE AND NONINFRINGEMENT. IN NO EVENT SHALL THE 
AUTHORS OR COPYRIGHT HOLDERS BE LIABLE FOR ANY CLAIM, DAMAGES OR OTHER 
LIABILITY, WHETHER IN AN ACTION OF CONTRACT, TORT OR OTHERWISE, ARISING FROM, 
OUT OF OR IN CONNECTION WITH THE SOFTWARE OR THE USE OR OTHER DEALINGS 
IN THE SOFTWARE.
*)
trigger := 0;
                    
END_ACTION

ACTION Init_active:
                      (*
Copyright (c) 2019 Manuel Goester, Michael Witt, Klaus Kammerer
Institute of Databases and Information Systems, Ulm University, Germany

Permission is hereby granted, free of charge, to any person obtaining a copy 
of this software and associated documentation files (the "Software"), to deal 
in the Software without restriction, including without limitation the rights 
to use, copy, modify, merge, publish, distribute, sublicense, and/or sell 
copies of the Software, and to permit persons to whom the Software is 
furnished to do so, subject to the following conditions:

The above copyright notice and this permission notice shall be included in 
all copies or substantial portions of the Software.

THE SOFTWARE IS PROVIDED "AS IS", WITHOUT WARRANTY OF ANY KIND, EXPRESS OR 
IMPLIED, INCLUDING BUT NOT LIMITED TO THE WARRANTIES OF MERCHANTABILITY, 
FITNESS FOR A PARTICULAR PURPOSE AND NONINFRINGEMENT. IN NO EVENT SHALL THE 
AUTHORS OR COPYRIGHT HOLDERS BE LIABLE FOR ANY CLAIM, DAMAGES OR OTHER 
LIABILITY, WHETHER IN AN ACTION OF CONTRACT, TORT OR OTHERWISE, ARISING FROM, 
OUT OF OR IN CONNECTION WITH THE SOFTWARE OR THE USE OR OTHER DEALINGS 
IN THE SOFTWARE.
*)
FUR.state := -1;
sawStopped := FALSE;
trigger := 0;
                    
END_ACTION

ACTION FUR_SUCCER_DOWN2_active:
                      (*
Copyright (c) 2019 Manuel Goester, Michael Witt, Klaus Kammerer
Institute of Databases and Information Systems, Ulm University, Germany

Permission is hereby granted, free of charge, to any person obtaining a copy 
of this software and associated documentation files (the "Software"), to deal 
in the Software without restriction, including without limitation the rights 
to use, copy, modify, merge, publish, distribute, sublicense, and/or sell 
copies of the Software, and to permit persons to whom the Software is 
furnished to do so, subject to the following conditions:

The above copyright notice and this permission notice shall be included in 
all copies or substantial portions of the Software.

THE SOFTWARE IS PROVIDED "AS IS", WITHOUT WARRANTY OF ANY KIND, EXPRESS OR 
IMPLIED, INCLUDING BUT NOT LIMITED TO THE WARRANTIES OF MERCHANTABILITY, 
FITNESS FOR A PARTICULAR PURPOSE AND NONINFRINGEMENT. IN NO EVENT SHALL THE 
AUTHORS OR COPYRIGHT HOLDERS BE LIABLE FOR ANY CLAIM, DAMAGES OR OTHER 
LIABILITY, WHETHER IN AN ACTION OF CONTRACT, TORT OR OTHERWISE, ARISING FROM, 
OUT OF OR IN CONNECTION WITH THE SOFTWARE OR THE USE OR OTHER DEALINGS 
IN THE SOFTWARE.
*)
IF FUR.sFurnanceSliderOutside THEN
	FUR.compressor := TRUE;
	FUR.valveLowering := TRUE;
	FUR.valveVacuum := FALSE;
	timer(IN:= TRUE, PT := T#1S);
	IF NOT(timer.Q = FALSE AND timer.IN) THEN
		timer(IN:= FALSE);
		FUR.valveLowering := FALSE;
		FUR.state := FUR_State.FUR_SUCCER_DOWN_AT_RD;
	END_IF
END_IF

                    
END_ACTION

ACTION FUR_SUCCER_DOWN_active:
                      (*
Copyright (c) 2019 Manuel Goester, Michael Witt, Klaus Kammerer
Institute of Databases and Information Systems, Ulm University, Germany

Permission is hereby granted, free of charge, to any person obtaining a copy 
of this software and associated documentation files (the "Software"), to deal 
in the Software without restriction, including without limitation the rights 
to use, copy, modify, merge, publish, distribute, sublicense, and/or sell 
copies of the Software, and to permit persons to whom the Software is 
furnished to do so, subject to the following conditions:

The above copyright notice and this permission notice shall be included in 
all copies or substantial portions of the Software.

THE SOFTWARE IS PROVIDED "AS IS", WITHOUT WARRANTY OF ANY KIND, EXPRESS OR 
IMPLIED, INCLUDING BUT NOT LIMITED TO THE WARRANTIES OF MERCHANTABILITY, 
FITNESS FOR A PARTICULAR PURPOSE AND NONINFRINGEMENT. IN NO EVENT SHALL THE 
AUTHORS OR COPYRIGHT HOLDERS BE LIABLE FOR ANY CLAIM, DAMAGES OR OTHER 
LIABILITY, WHETHER IN AN ACTION OF CONTRACT, TORT OR OTHERWISE, ARISING FROM, 
OUT OF OR IN CONNECTION WITH THE SOFTWARE OR THE USE OR OTHER DEALINGS 
IN THE SOFTWARE.
*)
timer(IN:= TRUE, PT := T#2S);
//sauger zum ofen
IF FUR.sFurnanceSliderOutside THEN
	FUR.compressor := TRUE;
	FUR.valveLowering := TRUE;
END_IF

IF NOT(timer.Q = FALSE AND timer.IN) THEN
	// reset timer
	timer(IN:= FALSE);
	// go to next step
	FUR.state := FUR_State.FUR_SUCCER_DOWN_AT_FUR;
END_IF
                    
END_ACTION

ACTION FUR_TO_CONVEYOR_active:
                      (*
Copyright (c) 2019 Manuel Goester, Michael Witt, Klaus Kammerer
Institute of Databases and Information Systems, Ulm University, Germany

Permission is hereby granted, free of charge, to any person obtaining a copy 
of this software and associated documentation files (the "Software"), to deal 
in the Software without restriction, including without limitation the rights 
to use, copy, modify, merge, publish, distribute, sublicense, and/or sell 
copies of the Software, and to permit persons to whom the Software is 
furnished to do so, subject to the following conditions:

The above copyright notice and this permission notice shall be included in 
all copies or substantial portions of the Software.

THE SOFTWARE IS PROVIDED "AS IS", WITHOUT WARRANTY OF ANY KIND, EXPRESS OR 
IMPLIED, INCLUDING BUT NOT LIMITED TO THE WARRANTIES OF MERCHANTABILITY, 
FITNESS FOR A PARTICULAR PURPOSE AND NONINFRINGEMENT. IN NO EVENT SHALL THE 
AUTHORS OR COPYRIGHT HOLDERS BE LIABLE FOR ANY CLAIM, DAMAGES OR OTHER 
LIABILITY, WHETHER IN AN ACTION OF CONTRACT, TORT OR OTHERWISE, ARISING FROM, 
OUT OF OR IN CONNECTION WITH THE SOFTWARE OR THE USE OR OTHER DEALINGS 
IN THE SOFTWARE.
*)
SM.currW.state := W_State.AT_FUR_ON_CONVEYOR;
SL.state := SL_State.W_RECEIVED;
IF NOT(FUR.sRaPosConveyorBelt) THEN
	FUR.mRaClockwise := TRUE;
ELSE
	FUR.mRaClockwise := FALSE;
	FUR.compressor := TRUE;
	FUR.valveSlider := TRUE;
END_IF

IF SL.lbEntry THEN
	FUR.mConveyorBeltForward := TRUE;
ELSE
	FUR.mConveyorBeltForward := FALSE;
	FUR.compressor := FALSE;
	FUR.valveSlider := FALSE;
	FUR.state := FUR_State.FUR_W_FINISHED_BACK_TO_DEFAULT;
END_IF
                    
END_ACTION

ACTION FUR_SUCCER_UP_active:
                      (*
Copyright (c) 2019 Manuel Goester, Michael Witt, Klaus Kammerer
Institute of Databases and Information Systems, Ulm University, Germany

Permission is hereby granted, free of charge, to any person obtaining a copy 
of this software and associated documentation files (the "Software"), to deal 
in the Software without restriction, including without limitation the rights 
to use, copy, modify, merge, publish, distribute, sublicense, and/or sell 
copies of the Software, and to permit persons to whom the Software is 
furnished to do so, subject to the following conditions:

The above copyright notice and this permission notice shall be included in 
all copies or substantial portions of the Software.

THE SOFTWARE IS PROVIDED "AS IS", WITHOUT WARRANTY OF ANY KIND, EXPRESS OR 
IMPLIED, INCLUDING BUT NOT LIMITED TO THE WARRANTIES OF MERCHANTABILITY, 
FITNESS FOR A PARTICULAR PURPOSE AND NONINFRINGEMENT. IN NO EVENT SHALL THE 
AUTHORS OR COPYRIGHT HOLDERS BE LIABLE FOR ANY CLAIM, DAMAGES OR OTHER 
LIABILITY, WHETHER IN AN ACTION OF CONTRACT, TORT OR OTHERWISE, ARISING FROM, 
OUT OF OR IN CONNECTION WITH THE SOFTWARE OR THE USE OR OTHER DEALINGS 
IN THE SOFTWARE.
*)
FUR.valveLowering := FALSE;
FUR.valveVacuum := TRUE; //hier, sonst wird kein vakuum erzeugt
SM.currW.state := W_State.AT_FUR_ATTACHED_TO_SUCCER;
FUR.state := FUR_State.FUR_SUCCER_UP_AT_FUR;
                    
END_ACTION

ACTION FUR_TO_DEFAULT_POS_active:
                      (*
Copyright (c) 2019 Manuel Goester, Michael Witt, Klaus Kammerer
Institute of Databases and Information Systems, Ulm University, Germany

Permission is hereby granted, free of charge, to any person obtaining a copy 
of this software and associated documentation files (the "Software"), to deal 
in the Software without restriction, including without limitation the rights 
to use, copy, modify, merge, publish, distribute, sublicense, and/or sell 
copies of the Software, and to permit persons to whom the Software is 
furnished to do so, subject to the following conditions:

The above copyright notice and this permission notice shall be included in 
all copies or substantial portions of the Software.

THE SOFTWARE IS PROVIDED "AS IS", WITHOUT WARRANTY OF ANY KIND, EXPRESS OR 
IMPLIED, INCLUDING BUT NOT LIMITED TO THE WARRANTIES OF MERCHANTABILITY, 
FITNESS FOR A PARTICULAR PURPOSE AND NONINFRINGEMENT. IN NO EVENT SHALL THE 
AUTHORS OR COPYRIGHT HOLDERS BE LIABLE FOR ANY CLAIM, DAMAGES OR OTHER 
LIABILITY, WHETHER IN AN ACTION OF CONTRACT, TORT OR OTHERWISE, ARISING FROM, 
OUT OF OR IN CONNECTION WITH THE SOFTWARE OR THE USE OR OTHER DEALINGS 
IN THE SOFTWARE.
*)
IF NOT(FUR.sFurnanceSliderOutside) THEN
	FUR.mFurnanceSliderOut := TRUE;
ELSE
	FUR.mFurnanceSliderOut := FALSE;
END_IF

IF NOT(FUR.sSuckerPosRa) THEN
	FUR.mSuckertoRa := TRUE;
ELSE
	FUR.mSuckertoRa := FALSE;
END_IF

IF NOT(FUR.sRaPosSucker) THEN
	FUR.mRaCClockwise := TRUE;
ELSE
	FUR.mRaCClockwise := FALSE;
END_IF

IF FUR.sSuckerPosRa AND FUR.sRaPosSucker AND FUR.sFurnanceSliderOutside THEN
	FUR.state := FUR_WAITING_FOR_W;
END_IF
                    
END_ACTION

ACTION FUR_WAIT_FOR_W_active:
                      (*
Copyright (c) 2019 Manuel Goester, Michael Witt, Klaus Kammerer
Institute of Databases and Information Systems, Ulm University, Germany

Permission is hereby granted, free of charge, to any person obtaining a copy 
of this software and associated documentation files (the "Software"), to deal 
in the Software without restriction, including without limitation the rights 
to use, copy, modify, merge, publish, distribute, sublicense, and/or sell 
copies of the Software, and to permit persons to whom the Software is 
furnished to do so, subject to the following conditions:

The above copyright notice and this permission notice shall be included in 
all copies or substantial portions of the Software.

THE SOFTWARE IS PROVIDED "AS IS", WITHOUT WARRANTY OF ANY KIND, EXPRESS OR 
IMPLIED, INCLUDING BUT NOT LIMITED TO THE WARRANTIES OF MERCHANTABILITY, 
FITNESS FOR A PARTICULAR PURPOSE AND NONINFRINGEMENT. IN NO EVENT SHALL THE 
AUTHORS OR COPYRIGHT HOLDERS BE LIABLE FOR ANY CLAIM, DAMAGES OR OTHER 
LIABILITY, WHETHER IN AN ACTION OF CONTRACT, TORT OR OTHERWISE, ARISING FROM, 
OUT OF OR IN CONNECTION WITH THE SOFTWARE OR THE USE OR OTHER DEALINGS 
IN THE SOFTWARE.
*)
// Workpiece passes the light barrier
IF NOT(FUR.lbFurnance) AND trigger < 2 THEN
	trigger := trigger + 1;
END_IF

// Workpiece passed light barrier
IF FUR.lbFurnance AND trigger >= 2 THEN
	FUR.state := FUR_State.FUR_LB_PASSED;
END_IF


                    
END_ACTION

ACTION FUR_BURN_active:
                      (*
Copyright (c) 2019 Manuel Goester, Michael Witt, Klaus Kammerer
Institute of Databases and Information Systems, Ulm University, Germany

Permission is hereby granted, free of charge, to any person obtaining a copy 
of this software and associated documentation files (the "Software"), to deal 
in the Software without restriction, including without limitation the rights 
to use, copy, modify, merge, publish, distribute, sublicense, and/or sell 
copies of the Software, and to permit persons to whom the Software is 
furnished to do so, subject to the following conditions:

The above copyright notice and this permission notice shall be included in 
all copies or substantial portions of the Software.

THE SOFTWARE IS PROVIDED "AS IS", WITHOUT WARRANTY OF ANY KIND, EXPRESS OR 
IMPLIED, INCLUDING BUT NOT LIMITED TO THE WARRANTIES OF MERCHANTABILITY, 
FITNESS FOR A PARTICULAR PURPOSE AND NONINFRINGEMENT. IN NO EVENT SHALL THE 
AUTHORS OR COPYRIGHT HOLDERS BE LIABLE FOR ANY CLAIM, DAMAGES OR OTHER 
LIABILITY, WHETHER IN AN ACTION OF CONTRACT, TORT OR OTHERWISE, ARISING FROM, 
OUT OF OR IN CONNECTION WITH THE SOFTWARE OR THE USE OR OTHER DEALINGS 
IN THE SOFTWARE.
*)
IF SM.currW.format.furEnabled THEN
	// open door and drive workpiece into furnance 
	IF FUR.state = FUR_State.FUR_LB_PASSED THEN
		FUR.compressor := TRUE;
		FUR.valveFurnanceDoor := TRUE;
		IF FUR.sFurnanceSliderInside = FALSE THEN
			FUR.mFurnanceSliderIn := TRUE;
		ELSE
			FUR.mFurnanceSliderIn := FALSE;
			FUR.state := FUR_State.FUR_WAGON_INSIDE;
		END_IF
	END_IF
	
	// burn
	IF FUR.state = FUR_State.FUR_WAGON_INSIDE THEN
		SM.currW.state := W_State.AT_FUR_IN_FUR;
		timer(IN:= TRUE, PT := SM.currW.format.furDuration);
		FUR.valveFurnanceDoor := FALSE;
		trigger := 0;
		
		// timer finished
		IF NOT(timer.Q = FALSE AND timer.IN) THEN
			timer(IN:= FALSE);
			FUR.compressor := TRUE;
			FUR.valveFurnanceDoor := TRUE;
			FUR.state := FUR_State.FUR_BURNED;
		END_IF
	END_IF
	
	// drive slider out
	IF FUR.state = FUR_State.FUR_BURNED THEN
		SM.currW.state := W_State.AT_FUR_IN_WAGON;
		IF FUR.sFurnanceSliderOutside = FALSE THEN
			FUR.mFurnanceSliderOut := TRUE;
		ELSE
			FUR.mFurnanceSliderOut := FALSE;
			FUR.state := FUR_State.FUR_WAGON_OUTSIDE;
		END_IF
	END_IF
	
	
	// bring succer to furnace
	IF NOT(FUR.sSuckerPosFF) AND (FUR.state = FUR_State.FUR_WAGON_INSIDE OR FUR.state = FUR_State.FUR_BURNED OR FUR.state = FUR_State.FUR_WAGON_OUTSIDE) THEN
		FUR.mSuckertoFurnance := TRUE;
	ELSE
		FUR.mSuckertoFurnance := FALSE;
	END_IF
	
	IF FUR.state = FUR_State.FUR_WAGON_OUTSIDE AND FUR.sSuckerPosFF THEN
		FUR.state := FUR_State.FUR_SUCCER_AT_FUR;
		FUR.mFurnanceSliderOut := FALSE;
		FUR.compressor := FALSE;
		FUR.valveFurnanceDoor := FALSE;
	END_IF
	
ELSE	
	// skip burning
	// bring succer to furnance
	IF NOT(FUR.sSuckerPosFF) THEN
		FUR.mSuckertoFurnance := TRUE;
	ELSE
		FUR.mSuckertoFurnance := FALSE;
		FUR.state := FUR_State.FUR_SUCCER_AT_FUR;
	END_IF
END_IF

                    
END_ACTION
END_PROGRAM

(* Adds a BatchJob to TC.BatchJobQueue Copyright (c) 2019 Manuel Goester, Michael Witt, Klaus Kammerer Institute of Databases and Information Systems, Ulm University, Germany Permission is hereby granted, free of charge, to any person obtaining a copy of this software and associated documentation files (the "Software"), to deal in the Software without restriction, including without limitation the rights to use, copy, modify, merge, publish, distribute, sublicense, and/or sell copies of the Software, and to permit persons to whom the Software is furnished to do so, subject to the following conditions: The above copyright notice and this permission notice shall be included in all copies or substantial portions of the Software. THE SOFTWARE IS PROVIDED "AS IS", WITHOUT WARRANTY OF ANY KIND, EXPRESS OR IMPLIED, INCLUDING BUT NOT LIMITED TO THE WARRANTIES OF MERCHANTABILITY, FITNESS FOR A PARTICULAR PURPOSE AND NONINFRINGEMENT. IN NO EVENT SHALL THE AUTHORS OR COPYRIGHT HOLDERS BE LIABLE FOR ANY CLAIM, DAMAGES OR OTHER LIABILITY, WHETHER IN AN ACTION OF CONTRACT, TORT OR OTHERWISE, ARISING FROM, OUT OF OR IN CONNECTION WITH THE SOFTWARE OR THE USE OR OTHER DEALINGS IN THE SOFTWARE. *)
FUNCTION addBatchJobToQueue : BOOL
  VAR_INPUT
    batchJob : BatchJob;  (* The BatchJob which will be added *)
  END_VAR

                  IF 1 <= TC.batchJobQueue.nextFreePos AND TC.batchJobQueue.nextFreePos <= 20 THEN
	TC.batchJobQueue.batchJobs[TC.batchJobQueue.nextFreePos] := batchJob;
	TC.batchJobQueue.nextFreePos := TC.batchJobQueue.nextFreePos + 1;
	TC.batchJobQueue.amountBatchJobs := TC.batchJobQueue.amountBatchJobs + 1;
	IF TC.batchJobQueue.amountBatchJobs = 20 THEN
		TC.batchJobQueue.full := TRUE;
	ELSE
		TC.batchJobQueue.full := FALSE;
	END_IF
	addBatchJobToQueue := TRUE;
ELSE
	// Batch Job Queue already full
	addBatchJobToQueue := FALSE;	
END_IF
RETURN;
                
END_FUNCTION

(* Constructor for Workpiece Copyright (c) 2019 Manuel Goester, Michael Witt, Klaus Kammerer Institute of Databases and Information Systems, Ulm University, Germany Permission is hereby granted, free of charge, to any person obtaining a copy of this software and associated documentation files (the "Software"), to deal in the Software without restriction, including without limitation the rights to use, copy, modify, merge, publish, distribute, sublicense, and/or sell copies of the Software, and to permit persons to whom the Software is furnished to do so, subject to the following conditions: The above copyright notice and this permission notice shall be included in all copies or substantial portions of the Software. THE SOFTWARE IS PROVIDED "AS IS", WITHOUT WARRANTY OF ANY KIND, EXPRESS OR IMPLIED, INCLUDING BUT NOT LIMITED TO THE WARRANTIES OF MERCHANTABILITY, FITNESS FOR A PARTICULAR PURPOSE AND NONINFRINGEMENT. IN NO EVENT SHALL THE AUTHORS OR COPYRIGHT HOLDERS BE LIABLE FOR ANY CLAIM, DAMAGES OR OTHER LIABILITY, WHETHER IN AN ACTION OF CONTRACT, TORT OR OTHERWISE, ARISING FROM, OUT OF OR IN CONNECTION WITH THE SOFTWARE OR THE USE OR OTHER DEALINGS IN THE SOFTWARE. *)
FUNCTION newWorkpiece : Workpiece
  VAR_INPUT
    color : STRING(7);  (* color of the workpiece: red, blue, white or unknown *)
    state : W_State;  (* state at start: 1ij, i = vertical pos in rack at begin, j = horizontal pos in rack at begin *)
    startPos : RackPos;
    endPos : RackPos;
    format : Format;  (* format for this workpiece *)
  END_VAR

                  newWorkpiece.color := color;
newWorkpiece.format := format;
newWorkpiece.startPos := startPos;
newWorkpiece.endPos := endPos;
newWorkpiece.sortingLinePos := -1;
newWorkpiece.linePos := 0;
newWorkpiece.state := state;
RETURN;
                
END_FUNCTION

PROGRAM SL_SINGLE_MODE
  VAR
    sl_fb : SL_FB;
    step : INT := 1;
    fin : BOOL;
  END_VAR

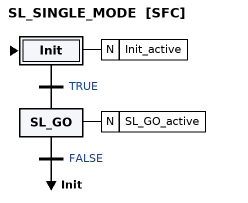
INITIAL_STEP Init:
  Init_active(N);
END_STEP
TRANSITION FROM Init TO SL_GO
  := TRUE;
END_TRANSITION
STEP SL_GO:
  SL_GO_active(N);
END_STEP
TRANSITION FROM SL_GO TO Init
  := FALSE;
END_TRANSITION

ACTION Init_active:
                      (*
Copyright (c) 2019 Manuel Goester, Michael Witt, Klaus Kammerer
Institute of Databases and Information Systems, Ulm University, Germany

Permission is hereby granted, free of charge, to any person obtaining a copy 
of this software and associated documentation files (the "Software"), to deal 
in the Software without restriction, including without limitation the rights 
to use, copy, modify, merge, publish, distribute, sublicense, and/or sell 
copies of the Software, and to permit persons to whom the Software is 
furnished to do so, subject to the following conditions:

The above copyright notice and this permission notice shall be included in 
all copies or substantial portions of the Software.

THE SOFTWARE IS PROVIDED "AS IS", WITHOUT WARRANTY OF ANY KIND, EXPRESS OR 
IMPLIED, INCLUDING BUT NOT LIMITED TO THE WARRANTIES OF MERCHANTABILITY, 
FITNESS FOR A PARTICULAR PURPOSE AND NONINFRINGEMENT. IN NO EVENT SHALL THE 
AUTHORS OR COPYRIGHT HOLDERS BE LIABLE FOR ANY CLAIM, DAMAGES OR OTHER 
LIABILITY, WHETHER IN AN ACTION OF CONTRACT, TORT OR OTHERWISE, ARISING FROM, 
OUT OF OR IN CONNECTION WITH THE SOFTWARE OR THE USE OR OTHER DEALINGS 
IN THE SOFTWARE.
*)
SL.state := SL_State.WAITING_FOR_W;
                    
END_ACTION

ACTION SL_GO_active:
                      (*
Copyright (c) 2019 Manuel Goester, Michael Witt, Klaus Kammerer
Institute of Databases and Information Systems, Ulm University, Germany

Permission is hereby granted, free of charge, to any person obtaining a copy 
of this software and associated documentation files (the "Software"), to deal 
in the Software without restriction, including without limitation the rights 
to use, copy, modify, merge, publish, distribute, sublicense, and/or sell 
copies of the Software, and to permit persons to whom the Software is 
furnished to do so, subject to the following conditions:

The above copyright notice and this permission notice shall be included in 
all copies or substantial portions of the Software.

THE SOFTWARE IS PROVIDED "AS IS", WITHOUT WARRANTY OF ANY KIND, EXPRESS OR 
IMPLIED, INCLUDING BUT NOT LIMITED TO THE WARRANTIES OF MERCHANTABILITY, 
FITNESS FOR A PARTICULAR PURPOSE AND NONINFRINGEMENT. IN NO EVENT SHALL THE 
AUTHORS OR COPYRIGHT HOLDERS BE LIABLE FOR ANY CLAIM, DAMAGES OR OTHER 
LIABILITY, WHETHER IN AN ACTION OF CONTRACT, TORT OR OTHERWISE, ARISING FROM, 
OUT OF OR IN CONNECTION WITH THE SOFTWARE OR THE USE OR OTHER DEALINGS 
IN THE SOFTWARE.
*)
CASE step OF
	1:
		IF SL.state = SL_State.W_RECEIVED THEN
			step := step + 1;
		END_IF
	2:
		IF NOT(fin) THEN
			sl_fb();
			fin := sl_fb.fin;
		ELSE
			// wait for VG to pick up w
			SL.state := SL_State.WAITING_FOR_VG_TO_PICK_UP_W;
			step := step + 1;
		END_IF
	3:
		// reset own pointers
		SL.bIdx := 0;
		SL.wIdx := 0;
		// reset fin
		fin := FALSE;
		step := 1;
		SL.state := SL_State.WAITING_FOR_W;
END_CASE
                    
END_ACTION
END_PROGRAM

(* Adds the workpiece w to the batchJobs queue, if there is a free place in the queue Copyright (c) 2019 Manuel Goester, Michael Witt, Klaus Kammerer Institute of Databases and Information Systems, Ulm University, Germany Permission is hereby granted, free of charge, to any person obtaining a copy of this software and associated documentation files (the "Software"), to deal in the Software without restriction, including without limitation the rights to use, copy, modify, merge, publish, distribute, sublicense, and/or sell copies of the Software, and to permit persons to whom the Software is furnished to do so, subject to the following conditions: The above copyright notice and this permission notice shall be included in all copies or substantial portions of the Software. THE SOFTWARE IS PROVIDED "AS IS", WITHOUT WARRANTY OF ANY KIND, EXPRESS OR IMPLIED, INCLUDING BUT NOT LIMITED TO THE WARRANTIES OF MERCHANTABILITY, FITNESS FOR A PARTICULAR PURPOSE AND NONINFRINGEMENT. IN NO EVENT SHALL THE AUTHORS OR COPYRIGHT HOLDERS BE LIABLE FOR ANY CLAIM, DAMAGES OR OTHER LIABILITY, WHETHER IN AN ACTION OF CONTRACT, TORT OR OTHERWISE, ARISING FROM, OUT OF OR IN CONNECTION WITH THE SOFTWARE OR THE USE OR OTHER DEALINGS IN THE SOFTWARE. *)
FUNCTION addWorkpieceToBatchJob : BOOL
  VAR_INPUT
    batchJob : BatchJob;  (* the batch job *)
    w : workpiece;  (* the workpiece to be added to the batch jobs queue *)
  END_VAR

                  IF batchJob.nextFreeWPos >= 1 AND batchJob.nextFreeWPos <= 9 THEN
	// free place available
	batchJob.workpieces[batchJob.nextFreeWPos] := w;
	batchJob.nextFreeWPos := batchJob.nextFreeWPos + 1;
	batchJob.batchSize := batchJob.batchSize + 1;
	AddWorkpieceToBatchJob := TRUE;
ELSE
	// queue full
	AddWorkpieceToBatchJob := FALSE;
END_IF
RETURN;
                
END_FUNCTION

PROGRAM VG_MULTI_MODE
  VAR
    fin : BOOL;
    step : INT := 1;
    timer : TON;
    sorting_line_pos : INT := -1;
    vg_move_to_pos : VG_MOVE_TO_POS;
    vg_move : VG_MOVE;
  END_VAR

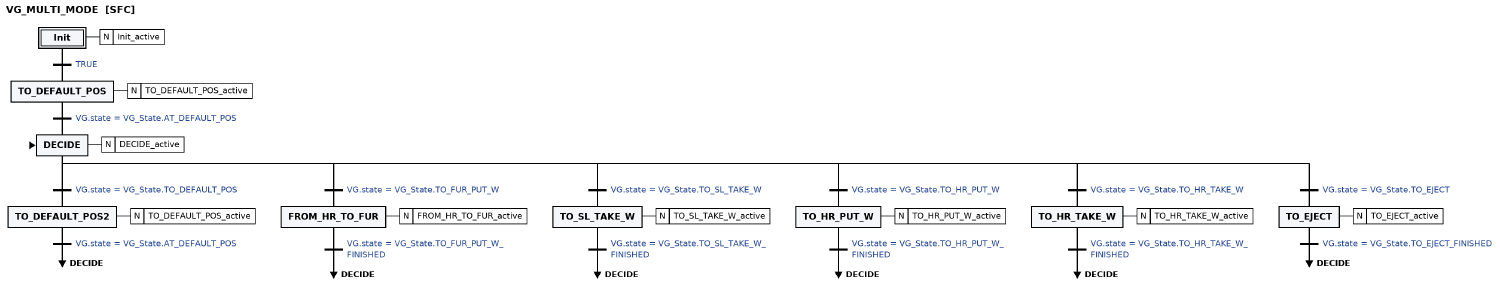
INITIAL_STEP Init:
  Init_active(N);
END_STEP
TRANSITION FROM Init TO TO_DEFAULT_POS
  := TRUE;
END_TRANSITION
STEP TO_DEFAULT_POS:
  TO_DEFAULT_POS_active(N);
END_STEP
TRANSITION FROM TO_DEFAULT_POS TO DECIDE
  := VG.state = VG_State.AT_DEFAULT_POS;
END_TRANSITION
STEP DECIDE:
  DECIDE_active(N);
END_STEP
TRANSITION FROM DECIDE TO TO_DEFAULT_POS2
  := VG.state = VG_State.TO_DEFAULT_POS;
END_TRANSITION
TRANSITION FROM DECIDE TO FROM_HR_TO_FUR
  := VG.state = VG_State.TO_FUR_PUT_W;
END_TRANSITION
TRANSITION FROM DECIDE TO TO_SL_TAKE_W
  := VG.state = VG_State.TO_SL_TAKE_W;
END_TRANSITION
TRANSITION FROM DECIDE TO TO_HR_PUT_W
  := VG.state = VG_State.TO_HR_PUT_W;
END_TRANSITION
TRANSITION FROM DECIDE TO TO_HR_TAKE_W
  := VG.state = VG_State.TO_HR_TAKE_W;
END_TRANSITION
TRANSITION FROM DECIDE TO TO_EJECT
  := VG.state = VG_State.TO_EJECT;
END_TRANSITION
STEP TO_DEFAULT_POS2:
  TO_DEFAULT_POS_active(N);
END_STEP
TRANSITION FROM TO_DEFAULT_POS2 TO DECIDE
  := VG.state = VG_State.AT_DEFAULT_POS;
END_TRANSITION
STEP FROM_HR_TO_FUR:
  FROM_HR_TO_FUR_active(N);
END_STEP
TRANSITION FROM FROM_HR_TO_FUR TO DECIDE
  := VG.state = VG_State.TO_FUR_PUT_W_FINISHED;
END_TRANSITION
STEP TO_SL_TAKE_W:
  TO_SL_TAKE_W_active(N);
END_STEP
TRANSITION FROM TO_SL_TAKE_W TO DECIDE
  := VG.state = VG_State.TO_SL_TAKE_W_FINISHED;
END_TRANSITION
STEP TO_HR_PUT_W:
  TO_HR_PUT_W_active(N);
END_STEP
TRANSITION FROM TO_HR_PUT_W TO DECIDE
  := VG.state = VG_State.TO_HR_PUT_W_FINISHED;
END_TRANSITION
STEP TO_HR_TAKE_W:
  TO_HR_TAKE_W_active(N);
END_STEP
TRANSITION FROM TO_HR_TAKE_W TO DECIDE
  := VG.state = VG_State.TO_HR_TAKE_W_FINISHED;
END_TRANSITION
STEP TO_EJECT:
  TO_EJECT_active(N);
END_STEP
TRANSITION FROM TO_EJECT TO DECIDE
  := VG.state = VG_State.TO_EJECT_FINISHED;
END_TRANSITION

ACTION TO_DEFAULT_POS_active:
                      (*
Copyright (c) 2019 Manuel Goester, Michael Witt, Klaus Kammerer
Institute of Databases and Information Systems, Ulm University, Germany

Permission is hereby granted, free of charge, to any person obtaining a copy 
of this software and associated documentation files (the "Software"), to deal 
in the Software without restriction, including without limitation the rights 
to use, copy, modify, merge, publish, distribute, sublicense, and/or sell 
copies of the Software, and to permit persons to whom the Software is 
furnished to do so, subject to the following conditions:

The above copyright notice and this permission notice shall be included in 
all copies or substantial portions of the Software.

THE SOFTWARE IS PROVIDED "AS IS", WITHOUT WARRANTY OF ANY KIND, EXPRESS OR 
IMPLIED, INCLUDING BUT NOT LIMITED TO THE WARRANTIES OF MERCHANTABILITY, 
FITNESS FOR A PARTICULAR PURPOSE AND NONINFRINGEMENT. IN NO EVENT SHALL THE 
AUTHORS OR COPYRIGHT HOLDERS BE LIABLE FOR ANY CLAIM, DAMAGES OR OTHER 
LIABILITY, WHETHER IN AN ACTION OF CONTRACT, TORT OR OTHERWISE, ARISING FROM, 
OUT OF OR IN CONNECTION WITH THE SOFTWARE OR THE USE OR OTHER DEALINGS 
IN THE SOFTWARE.
*)
// Brings VG to its default pos where sVertical = sHorizontal = sRotation = TRUE
// 1. y-Axis 2. z-Axis 3. rotation
IF NOT(VG.sVertical) THEN
	VG.mVerticalUp := TRUE;
ELSE
	VG.mVerticalUp := FALSE;
	// reset position counter
	VG.cY := 0;
	IF NOT(VG.sHorizontal) THEN
		VG.mHorizontalBackward := TRUE;
	ELSE
		VG.mHorizontalBackward := FALSE;
		// reset position counter
		VG.cX := 0;
		IF NOT(VG.sRotation) THEN
			VG.mRotationClockwise := TRUE;
		ELSE
			VG.mRotationClockwise := FALSE;
			// reset position counter
			VG.cZ := 0;
			
			// wait for 0.5 sec
			timer(IN:= TRUE, PT := T#0.5S);
			IF NOT(timer.Q = FALSE AND timer.IN) THEN
				timer(IN:=FALSE);
				
				// default pos reached
				VG.state := VG_State.AT_DEFAULT_POS;
			END_IF
		END_IF
	END_IF
END_IF
                    
END_ACTION

ACTION DECIDE_active:
                      (*
Copyright (c) 2019 Manuel Goester, Michael Witt, Klaus Kammerer
Institute of Databases and Information Systems, Ulm University, Germany

Permission is hereby granted, free of charge, to any person obtaining a copy 
of this software and associated documentation files (the "Software"), to deal 
in the Software without restriction, including without limitation the rights 
to use, copy, modify, merge, publish, distribute, sublicense, and/or sell 
copies of the Software, and to permit persons to whom the Software is 
furnished to do so, subject to the following conditions:

The above copyright notice and this permission notice shall be included in 
all copies or substantial portions of the Software.

THE SOFTWARE IS PROVIDED "AS IS", WITHOUT WARRANTY OF ANY KIND, EXPRESS OR 
IMPLIED, INCLUDING BUT NOT LIMITED TO THE WARRANTIES OF MERCHANTABILITY, 
FITNESS FOR A PARTICULAR PURPOSE AND NONINFRINGEMENT. IN NO EVENT SHALL THE 
AUTHORS OR COPYRIGHT HOLDERS BE LIABLE FOR ANY CLAIM, DAMAGES OR OTHER 
LIABILITY, WHETHER IN AN ACTION OF CONTRACT, TORT OR OTHERWISE, ARISING FROM, 
OUT OF OR IN CONNECTION WITH THE SOFTWARE OR THE USE OR OTHER DEALINGS 
IN THE SOFTWARE.
*)
IF VG.state = VG_State.AT_HR THEN
	// this can happen if the batch job before was a single mode batch job. Then VG is already AT HR and is not in ready state
	VG.state := VG_State.TO_HR_TAKE_W;
ELSIF VG.state = VG_State.READY AND (HR.state = HR_State.GET_W AND HR.currW.state <> W_State.NULL) THEN
	// go to HR and take w
	VG.state := VG_State.TO_HR_TAKE_W;
ELSIF VG.state = VG_State.READY AND (NOT(SL.lbWhite) OR NOT(SL.lbRed) OR NOT(SL.lbBlue)) AND SL.currW.state <> W_State.NULL AND (NOT(HR.decidedToTakeANewW) OR HR.currW.state = W_State.NULL) THEN
	// go to SL and take w
	// bend VG pointers to workpiece being picked up
	VG.bIdx := SL.bIdx;
	VG.wIdx := SL.wIdx;
	VG.currW := TC.batchJobQueue.batchJobs[VG.bIdx].workpieces[VG.wIdx];
	VG.state := VG_State.TO_SL_TAKE_W;
ELSIF VG.state = VG_State.TO_SL_TAKE_W_FINISHED THEN
	// reset SL pointers
	SL.bIdx := 0;
	SL.wIdx := 0;
	SL.currW := TC.nullW;
	// at SL, w taken, decide if going to EJECT or HR
	IF VG.currW.format.ejectEnabled THEN
		// go to eject point and eject w
		VG.state := VG_State.TO_EJECT;
	ELSE
		// go to HR and put down w
		VG.state := VG_State.TO_HR_PUT_W;
	END_IF
ELSIF VG.state = VG_State.TO_HR_TAKE_W_FINISHED THEN
	// at HR, w taken, decide if going to FUR or EJECT
	IF VG.currW.format.ejectEnabled AND NOT(VG.currW.format.colorCheckEnabled OR VG.currW.format.furEnabled OR VG.currW.format.sawEnabled) THEN
		// go to eject point and eject w
		VG.state := VG_State.TO_EJECT;
	ELSE
		// go to FUR and put down w
		// but only if FUR-succer is at its default pos
		IF FUR.sSuckerPosRa THEN
			VG.state := VG_State.TO_FUR_PUT_W;
		END_IF
	END_IF
ELSIF VG.state = VG_State.TO_EJECT_FINISHED OR VG.state = VG_State.TO_FUR_PUT_W_FINISHED OR  VG.state = VG_State.TO_HR_PUT_W_FINISHED THEN
	// eject or putting w to FUR finished, back to default position for calibrating axes
	// likewise if VG put down w at HR
	VG.state := VG_State.TO_DEFAULT_POS;
ELSIF VG.state = VG_State.AT_DEFAULT_POS THEN
	// state = ready if VG is at default pos or if VG put down a w at HR --> VG is ready for next w
	VG.state := VG_state.READY;
	// reset own pointers
	VG.bIdx := 0;
	VG.wIdx := 0;
	VG.currW := TC.nullW;
END_IF
                    
END_ACTION

ACTION FROM_HR_TO_FUR_active:
                      (*
Copyright (c) 2019 Manuel Goester, Michael Witt, Klaus Kammerer
Institute of Databases and Information Systems, Ulm University, Germany

Permission is hereby granted, free of charge, to any person obtaining a copy 
of this software and associated documentation files (the "Software"), to deal 
in the Software without restriction, including without limitation the rights 
to use, copy, modify, merge, publish, distribute, sublicense, and/or sell 
copies of the Software, and to permit persons to whom the Software is 
furnished to do so, subject to the following conditions:

The above copyright notice and this permission notice shall be included in 
all copies or substantial portions of the Software.

THE SOFTWARE IS PROVIDED "AS IS", WITHOUT WARRANTY OF ANY KIND, EXPRESS OR 
IMPLIED, INCLUDING BUT NOT LIMITED TO THE WARRANTIES OF MERCHANTABILITY, 
FITNESS FOR A PARTICULAR PURPOSE AND NONINFRINGEMENT. IN NO EVENT SHALL THE 
AUTHORS OR COPYRIGHT HOLDERS BE LIABLE FOR ANY CLAIM, DAMAGES OR OTHER 
LIABILITY, WHETHER IN AN ACTION OF CONTRACT, TORT OR OTHERWISE, ARISING FROM, 
OUT OF OR IN CONNECTION WITH THE SOFTWARE OR THE USE OR OTHER DEALINGS 
IN THE SOFTWARE.
*)
CASE step OF
	1:
		// x and z axis: move to FUR
		IF NOT(fin) THEN
			vg_move_to_pos(x := 131, y := 0, z := 137);
			fin := vg_move_to_pos.fin;
		ELSE
			fin := FALSE;
			step := step + 1;
		END_IF
	2:
		// y axis: move to FUR
		IF NOT(fin) THEN
			vg_move_to_pos(x := 131, y := 85, z := 137);
			fin := vg_move_to_pos.fin;
		ELSE
			fin := FALSE;
			step := step + 1;
		END_IF
	3:
		// open ventil to put down w onto waggon
		VG.valve := FALSE;
		step := step + 1;
	4:
		// wait 1 second to get sure w is not succed anymore
		timer(IN:= TRUE, PT:= T#1S);
		IF NOT(timer.Q = FALSE AND timer.IN) THEN
			// reset timer
			timer(IN:= FALSE);
			step := step + 1;
		END_IF
	5:
		// y axis: go up as far as possible
		IF NOT(VG.sVertical) THEN
			VG.mVerticalUp := TRUE;
		ELSE
			VG.mVerticalUp := FALSE;
			// reset y axis counter
			VG.cY := 0;
			// reset step counter
			step := 1;
			// bend FUR-Burner pointers to current workpiece of VG
			FUR.bIdxBurner := VG.bIdx;
			FUR.wIdxBurner := VG.wIdx;
			FUR.currWBurner := TC.batchJobQueue.batchJobs[FUR.bIdxBurner].workpieces[FUR.wIdxBurner];
			// finished
			VG.state := VG_State.TO_FUR_PUT_W_FINISHED;
		END_IF
	6:
	
END_CASE
                    
END_ACTION

ACTION TO_SL_TAKE_W_active:
                      (*
Copyright (c) 2019 Manuel Goester, Michael Witt, Klaus Kammerer
Institute of Databases and Information Systems, Ulm University, Germany

Permission is hereby granted, free of charge, to any person obtaining a copy 
of this software and associated documentation files (the "Software"), to deal 
in the Software without restriction, including without limitation the rights 
to use, copy, modify, merge, publish, distribute, sublicense, and/or sell 
copies of the Software, and to permit persons to whom the Software is 
furnished to do so, subject to the following conditions:

The above copyright notice and this permission notice shall be included in 
all copies or substantial portions of the Software.

THE SOFTWARE IS PROVIDED "AS IS", WITHOUT WARRANTY OF ANY KIND, EXPRESS OR 
IMPLIED, INCLUDING BUT NOT LIMITED TO THE WARRANTIES OF MERCHANTABILITY, 
FITNESS FOR A PARTICULAR PURPOSE AND NONINFRINGEMENT. IN NO EVENT SHALL THE 
AUTHORS OR COPYRIGHT HOLDERS BE LIABLE FOR ANY CLAIM, DAMAGES OR OTHER 
LIABILITY, WHETHER IN AN ACTION OF CONTRACT, TORT OR OTHERWISE, ARISING FROM, 
OUT OF OR IN CONNECTION WITH THE SOFTWARE OR THE USE OR OTHER DEALINGS 
IN THE SOFTWARE.
*)
CASE step OF
	1:
		IF NOT(SL.currW.format.ejectEnabled) THEN
			// set flag to inform HR that VG is taking a w to bring it back to HR
			VG.storeW := TRUE;
			//VG.bIdx := SL.bIdx;
			//VG.wIdx := SL.wIdx;
			//VG.currW := TC.batchJobQueue.batchJobs[VG.bIdx].workpieces[VG.wIdx];
		END_IF
		// select sorting line pos
		IF 	TC.batchJobQueue.batchJobs[SL.bIdx].workpieces[SL.wIdx].format.colorCheckEnabled THEN
			IF TC.batchJobQueue.batchJobs[SL.bIdx].workpieces[SL.wIdx].color = 'white' AND NOT(SL.lbWhite) THEN
				sorting_line_pos := 1;
			ELSIF TC.batchJobQueue.batchJobs[SL.bIdx].workpieces[SL.wIdx].color = 'red' AND NOT(SL.lbRed) THEN
				sorting_line_pos := 2;
			ELSIF TC.batchJobQueue.batchJobs[SL.bIdx].workpieces[SL.wIdx].color = 'blue' AND NOT(SL.lbBlue) THEN
				sorting_line_pos := 3;
			END_IF
		ELSE
			// when color was not checked
			sorting_line_pos := 1;
		END_IF
		step := step + 1;
	2:
		// x and z axis: move to SL
		IF NOT(fin) THEN
			CASE sorting_line_pos OF
				1:
					vg_move_to_pos(x := 58, y := 0, z := 69);
				2:
					vg_move_to_pos(x := 63, y := 0, z := 57);
				3:
					vg_move_to_pos(x := 87, y := 0, z := 47);
			END_CASE
		fin := vg_move_to_pos.fin;
		ELSE
			fin := FALSE;
			step := step + 1;
		END_IF
	3:
		// y axis: move to SL
		IF NOT(fin) THEN
			CASE sorting_line_pos OF
				1:
					vg_move_to_pos(x := 58, y := 125, z := 69);
				2:
					vg_move_to_pos(x := 63, y := 125, z := 57);
				3:
					vg_move_to_pos(x := 87, y := 125, z := 47);
			END_CASE
		fin := vg_move_to_pos.fin;
		ELSE
			fin := FALSE;
			step := step + 1;
		END_IF
	4:
		// succ workpiece at SL
		VG.valve := TRUE;
		timer(IN:= TRUE, PT:= T#2S);
		IF timer.Q = FALSE AND timer.IN THEN
			// go
			VG.compressor := TRUE;
		ELSE
			// stop
			VG.compressor := FALSE;
			// reset timer
			timer(IN:= FALSE);
			step := step + 1;
		END_IF
	5:
		// y axis: go up as far as possible
		IF NOT(VG.sVertical) THEN
			VG.mVerticalUp := TRUE;
		ELSE
			VG.mVerticalUp := FALSE;
			// reset y axis counter
			VG.cY := 0;
			// reset step counter
			step := 1;
			// reset sorting line pos
			sorting_line_pos := -1;
			// finished
			VG.state := VG_State.TO_SL_TAKE_W_FINISHED;
		END_IF
END_CASE
                    
END_ACTION

ACTION TO_HR_PUT_W_active:
                      (*
Copyright (c) 2019 Manuel Goester, Michael Witt, Klaus Kammerer
Institute of Databases and Information Systems, Ulm University, Germany

Permission is hereby granted, free of charge, to any person obtaining a copy 
of this software and associated documentation files (the "Software"), to deal 
in the Software without restriction, including without limitation the rights 
to use, copy, modify, merge, publish, distribute, sublicense, and/or sell 
copies of the Software, and to permit persons to whom the Software is 
furnished to do so, subject to the following conditions:

The above copyright notice and this permission notice shall be included in 
all copies or substantial portions of the Software.

THE SOFTWARE IS PROVIDED "AS IS", WITHOUT WARRANTY OF ANY KIND, EXPRESS OR 
IMPLIED, INCLUDING BUT NOT LIMITED TO THE WARRANTIES OF MERCHANTABILITY, 
FITNESS FOR A PARTICULAR PURPOSE AND NONINFRINGEMENT. IN NO EVENT SHALL THE 
AUTHORS OR COPYRIGHT HOLDERS BE LIABLE FOR ANY CLAIM, DAMAGES OR OTHER 
LIABILITY, WHETHER IN AN ACTION OF CONTRACT, TORT OR OTHERWISE, ARISING FROM, 
OUT OF OR IN CONNECTION WITH THE SOFTWARE OR THE USE OR OTHER DEALINGS 
IN THE SOFTWARE.
*)
CASE step OF
	1:
		// x and z axis: move to HR
		IF NOT(fin) THEN
			vg_move_to_pos(x := 27, y := 0, z := 206);
			fin := vg_move_to_pos.fin;
		ELSE
			fin := FALSE;
			step := step + 1;
		END_IF
	2:
		// box without workpiece arrived, wait 0.5 sec to be sure
		IF NOT(HR.lbOut) AND HR.state = HR_State.WAIT_FOR_VG_TO_BRING_W THEN
			timer(IN:= TRUE, PT:= T#0.5S);
			IF NOT(timer.Q = FALSE AND timer.IN) THEN
				timer(IN:= FALSE);
				step := step + 1;
			END_IF
		END_IF
	3:
		// y axis: move down at HR
		IF NOT(fin) THEN
			vg_move_to_pos(x:=27, y:=40, z:=206);
			fin := vg_move_to_pos.fin;
		ELSE
			fin := FALSE;
			step := step + 1;
		END_IF
	4:
		// open ventil
		VG.valve := FALSE;
		step := step + 1;
	5:
		timer(IN:= TRUE, PT:= T#1S);
		IF NOT(timer.Q = FALSE AND timer.IN) THEN
			// reset timer
			timer(IN:= FALSE);
			// go to next step
			step := step + 1;
		END_IF
	6:
		// y axis: go up as far as possible
		IF NOT(VG.sVertical) THEN
			VG.mVerticalUp := TRUE;
		ELSE
			VG.mVerticalUp := FALSE;
			// reset y axis counter
			VG.cY := 0;
			// reset step counter
			step := 1;
			// finished
			VG.state := VG_State.TO_HR_PUT_W_FINISHED;
		END_IF
END_CASE
                    
END_ACTION

ACTION TO_HR_TAKE_W_active:
                      (*
Copyright (c) 2019 Manuel Goester, Michael Witt, Klaus Kammerer
Institute of Databases and Information Systems, Ulm University, Germany

Permission is hereby granted, free of charge, to any person obtaining a copy 
of this software and associated documentation files (the "Software"), to deal 
in the Software without restriction, including without limitation the rights 
to use, copy, modify, merge, publish, distribute, sublicense, and/or sell 
copies of the Software, and to permit persons to whom the Software is 
furnished to do so, subject to the following conditions:

The above copyright notice and this permission notice shall be included in 
all copies or substantial portions of the Software.

THE SOFTWARE IS PROVIDED "AS IS", WITHOUT WARRANTY OF ANY KIND, EXPRESS OR 
IMPLIED, INCLUDING BUT NOT LIMITED TO THE WARRANTIES OF MERCHANTABILITY, 
FITNESS FOR A PARTICULAR PURPOSE AND NONINFRINGEMENT. IN NO EVENT SHALL THE 
AUTHORS OR COPYRIGHT HOLDERS BE LIABLE FOR ANY CLAIM, DAMAGES OR OTHER 
LIABILITY, WHETHER IN AN ACTION OF CONTRACT, TORT OR OTHERWISE, ARISING FROM, 
OUT OF OR IN CONNECTION WITH THE SOFTWARE OR THE USE OR OTHER DEALINGS 
IN THE SOFTWARE.
*)
CASE step OF
	1:
		// x and z axis: move to HR
		IF NOT(fin) THEN
			vg_move_to_pos(x := 27, y := 0, z := 206);
			fin := vg_move_to_pos.fin;
		ELSE
			fin := FALSE;
			step := step + 1;
		END_IF
	2:
		IF NOT(HR.lbOut) THEN
			// box with workpiece arrived, wait 0.5 sec to be sure
			timer(IN:= TRUE, PT:= T#0.5S);
			IF NOT(timer.Q = FALSE AND timer.IN) THEN
				timer(IN:= FALSE);
				step := step + 1;
			END_IF		
		END_IF
	3:
		// y axis: move down at HR
		IF NOT(fin) THEN
			vg_move_to_pos(x:=27, y:=40, z:=206);
			fin := vg_move_to_pos.fin;
		ELSE
			fin := FALSE;
			step := step + 1;
		END_IF
	4:
		// succ w at HR
		VG.valve := TRUE;
		timer(IN:= TRUE, PT:= T#2S);
		IF timer.Q = FALSE AND timer.IN THEN
			// go
			VG.compressor := TRUE;
		ELSE
			// stop
			VG.compressor := FALSE;
			// reset timer
			timer(IN:= FALSE);
			step := step + 1;
		END_IF	
	5:
		// y axis: go up as far as possible
		IF NOT(VG.sVertical) THEN
			VG.mVerticalUp := TRUE;
		ELSE
			VG.mVerticalUp := FALSE;
			// reset y axis counter
			VG.cY := 0;
			// reset step counter
			step := 1;
			// finished
			VG.state := VG_State.TO_HR_TAKE_W_FINISHED;
		END_IF
END_CASE
                    
END_ACTION

ACTION TO_EJECT_active:
                      (*
Copyright (c) 2019 Manuel Goester, Michael Witt, Klaus Kammerer
Institute of Databases and Information Systems, Ulm University, Germany

Permission is hereby granted, free of charge, to any person obtaining a copy 
of this software and associated documentation files (the "Software"), to deal 
in the Software without restriction, including without limitation the rights 
to use, copy, modify, merge, publish, distribute, sublicense, and/or sell 
copies of the Software, and to permit persons to whom the Software is 
furnished to do so, subject to the following conditions:

The above copyright notice and this permission notice shall be included in 
all copies or substantial portions of the Software.

THE SOFTWARE IS PROVIDED "AS IS", WITHOUT WARRANTY OF ANY KIND, EXPRESS OR 
IMPLIED, INCLUDING BUT NOT LIMITED TO THE WARRANTIES OF MERCHANTABILITY, 
FITNESS FOR A PARTICULAR PURPOSE AND NONINFRINGEMENT. IN NO EVENT SHALL THE 
AUTHORS OR COPYRIGHT HOLDERS BE LIABLE FOR ANY CLAIM, DAMAGES OR OTHER 
LIABILITY, WHETHER IN AN ACTION OF CONTRACT, TORT OR OTHERWISE, ARISING FROM, 
OUT OF OR IN CONNECTION WITH THE SOFTWARE OR THE USE OR OTHER DEALINGS 
IN THE SOFTWARE.
*)
CASE step OF
	1:
		// x and z axis: move to EJECT
		IF NOT(fin) THEN
			IF VG.currW.color = 'white' THEN
				// go to eject point 1
				vg_move_to_pos(x := 25, y := 0, z := 2);
			ELSIF VG.currW.color = 'red' THEN
				// go to eject point 2
				vg_move_to_pos(x := 30, y := 0, z := 15);
			ELSIF VG.currW.color = 'blue' THEN
				// go to eject point 3
				vg_move_to_pos(x := 49, y := 0, z := 23);
			ELSE
				// if color 'unknown' then eject to white eject point
				// go to eject point 1
				vg_move_to_pos(x := 25, y := 0, z := 2);
			END_IF
			fin := vg_move_to_pos.fin;
		ELSE
			fin := FALSE;
			step := step + 1;
		END_IF
	2:
		// x and z axis: move to EJECT
		IF NOT(fin) THEN
			IF VG.currW.color = 'white' THEN
				// go to eject point 1
				vg_move_to_pos(x := 25, y := 133, z := 2);
			ELSIF VG.currW.color = 'red' THEN
				// go to eject point 2
				vg_move_to_pos(x := 30, y := 133, z := 15);
			ELSIF VG.currW.color = 'blue' THEN
				// go to eject point 3
				vg_move_to_pos(x := 49, y := 133, z := 23);
			ELSE
				// if color 'unknown' then eject to white eject point
				// go to eject point 1
				vg_move_to_pos(x := 25, y := 133, z := 2);
			END_IF
			fin := vg_move_to_pos.fin;
		ELSE
			fin := FALSE;
			step := step + 1;
		END_IF
	3:
		// open valve to drop w
		VG.valve := FALSE;
		timer(IN:= TRUE, PT:= T#1S);
		IF NOT(timer.Q = FALSE AND timer.IN) THEN
			// reset timer
			timer(IN:= FALSE);
			// reset step counter
			step := 1;
			// finished
			VG.state := VG_State.TO_EJECT_FINISHED;
		END_IF
END_CASE
                    
END_ACTION

ACTION Init_active:
                      (*
Copyright (c) 2019 Manuel Goester, Michael Witt, Klaus Kammerer
Institute of Databases and Information Systems, Ulm University, Germany

Permission is hereby granted, free of charge, to any person obtaining a copy 
of this software and associated documentation files (the "Software"), to deal 
in the Software without restriction, including without limitation the rights 
to use, copy, modify, merge, publish, distribute, sublicense, and/or sell 
copies of the Software, and to permit persons to whom the Software is 
furnished to do so, subject to the following conditions:

The above copyright notice and this permission notice shall be included in 
all copies or substantial portions of the Software.

THE SOFTWARE IS PROVIDED "AS IS", WITHOUT WARRANTY OF ANY KIND, EXPRESS OR 
IMPLIED, INCLUDING BUT NOT LIMITED TO THE WARRANTIES OF MERCHANTABILITY, 
FITNESS FOR A PARTICULAR PURPOSE AND NONINFRINGEMENT. IN NO EVENT SHALL THE 
AUTHORS OR COPYRIGHT HOLDERS BE LIABLE FOR ANY CLAIM, DAMAGES OR OTHER 
LIABILITY, WHETHER IN AN ACTION OF CONTRACT, TORT OR OTHERWISE, ARISING FROM, 
OUT OF OR IN CONNECTION WITH THE SOFTWARE OR THE USE OR OTHER DEALINGS 
IN THE SOFTWARE.
*)
step := 1;
                    
END_ACTION
END_PROGRAM

PROGRAM TC_POU
  VAR
    started : BOOL;  (* true if user pressed start button *)
    batch_job_available : BOOL := FALSE;  (* true if theres a batch job waiting to be executed *)
    fin : BOOL;
    Copyright : INT;
  END_VAR

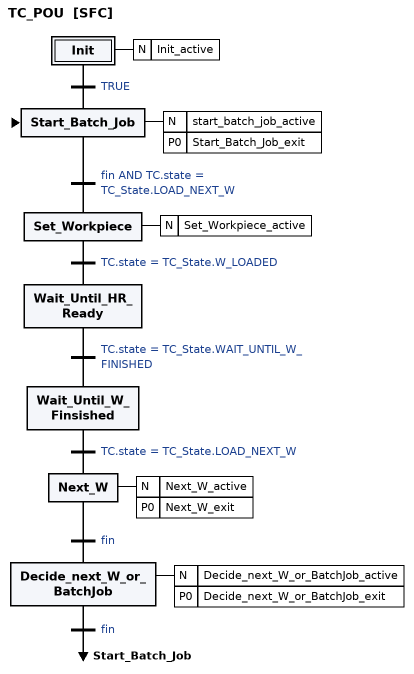
INITIAL_STEP Init:
  Init_active(N);
END_STEP
TRANSITION FROM Init TO Start_Batch_Job
  := TRUE;
END_TRANSITION
STEP Start_Batch_Job:
  start_batch_job_active(N);
  Start_Batch_Job_exit(P0);
END_STEP
TRANSITION FROM Start_Batch_Job TO Set_Workpiece
  := fin AND TC.state = TC_State.LOAD_NEXT_W;
END_TRANSITION
STEP Set_Workpiece:
  Set_Workpiece_active(N);
END_STEP
TRANSITION FROM Set_Workpiece TO Wait_Until_HR_Ready
  := TC.state = TC_State.W_LOADED;
END_TRANSITION
STEP Wait_Until_HR_Ready:
END_STEP
TRANSITION FROM Wait_Until_HR_Ready TO Wait_Until_W_Finsished
  := TC.state = TC_State.WAIT_UNTIL_W_FINISHED;
END_TRANSITION
STEP Wait_Until_W_Finsished:
END_STEP
TRANSITION FROM Wait_Until_W_Finsished TO Next_W
  := TC.state = TC_State.LOAD_NEXT_W;
END_TRANSITION
STEP Next_W:
  Next_W_active(N);
  Next_W_exit(P0);
END_STEP
TRANSITION FROM Next_W TO Decide_next_W_or_BatchJob
  := fin;
END_TRANSITION
STEP Decide_next_W_or_BatchJob:
  Decide_next_W_or_BatchJob_active(N);
  Decide_next_W_or_BatchJob_exit(P0);
END_STEP
TRANSITION FROM Decide_next_W_or_BatchJob TO Start_Batch_Job
  := fin;
END_TRANSITION

ACTION Decide_next_W_or_BatchJob_active:
                      (*
Copyright (c) 2019 Manuel Goester, Michael Witt, Klaus Kammerer
Institute of Databases and Information Systems, Ulm University, Germany

Permission is hereby granted, free of charge, to any person obtaining a copy 
of this software and associated documentation files (the "Software"), to deal 
in the Software without restriction, including without limitation the rights 
to use, copy, modify, merge, publish, distribute, sublicense, and/or sell 
copies of the Software, and to permit persons to whom the Software is 
furnished to do so, subject to the following conditions:

The above copyright notice and this permission notice shall be included in 
all copies or substantial portions of the Software.

THE SOFTWARE IS PROVIDED "AS IS", WITHOUT WARRANTY OF ANY KIND, EXPRESS OR 
IMPLIED, INCLUDING BUT NOT LIMITED TO THE WARRANTIES OF MERCHANTABILITY, 
FITNESS FOR A PARTICULAR PURPOSE AND NONINFRINGEMENT. IN NO EVENT SHALL THE 
AUTHORS OR COPYRIGHT HOLDERS BE LIABLE FOR ANY CLAIM, DAMAGES OR OTHER 
LIABILITY, WHETHER IN AN ACTION OF CONTRACT, TORT OR OTHERWISE, ARISING FROM, 
OUT OF OR IN CONNECTION WITH THE SOFTWARE OR THE USE OR OTHER DEALINGS 
IN THE SOFTWARE.
*)
IF NOT(fin) THEN
	IF TC.batchJobQueue.batchJobs[TC.currBatchJobIdx].nextNotProcessedIdx > TC.batchJobQueue.batchJobs[TC.currBatchJobIdx].batchSize THEN
		IF SM.currW.state = 0 AND HR.bIdx = 0 AND VG.bIdx = 0 AND FUR.bIdxBurner = 0 AND FUR.bIdxSuccer = 0 AND FUR.bIdxSaw = 0 AND SL.bIdx = 0 THEN
			// there is no new workpiece in current BatchJob and all maschines finished processing --> BatchJob finished
			TC.batchJobQueue.batchJobs[TC.currBatchJobIdx].state := BatchJobState.FINISHED;
			// delete finished BatchJob
			TC.batchJobQueue.batchJobs[TC.currBatchJobIdx] := TC.nullB;
			// update counter of BatchJobs in queue
			TC.batchJobQueue.amountBatchJobs := TC.batchJobQueue.amountBatchJobs - 1;
			// start next batch job if there is one
			TC.currBatchJobIdx := TC.currBatchJobIdx + 1;
			IF TC.currBatchJobIdx > 20 THEN
				TC.currBatchJobIdx := 1;
			END_IF
			fin := TRUE;
		END_IF
	ELSE
		// batch job not finished --> execute steps for next workpiece
		fin := TRUE;
	END_IF
END_IF
                    
END_ACTION

ACTION Set_Workpiece_active:
                      (*
Copyright (c) 2019 Manuel Goester, Michael Witt, Klaus Kammerer
Institute of Databases and Information Systems, Ulm University, Germany

Permission is hereby granted, free of charge, to any person obtaining a copy 
of this software and associated documentation files (the "Software"), to deal 
in the Software without restriction, including without limitation the rights 
to use, copy, modify, merge, publish, distribute, sublicense, and/or sell 
copies of the Software, and to permit persons to whom the Software is 
furnished to do so, subject to the following conditions:

The above copyright notice and this permission notice shall be included in 
all copies or substantial portions of the Software.

THE SOFTWARE IS PROVIDED "AS IS", WITHOUT WARRANTY OF ANY KIND, EXPRESS OR 
IMPLIED, INCLUDING BUT NOT LIMITED TO THE WARRANTIES OF MERCHANTABILITY, 
FITNESS FOR A PARTICULAR PURPOSE AND NONINFRINGEMENT. IN NO EVENT SHALL THE 
AUTHORS OR COPYRIGHT HOLDERS BE LIABLE FOR ANY CLAIM, DAMAGES OR OTHER 
LIABILITY, WHETHER IN AN ACTION OF CONTRACT, TORT OR OTHERWISE, ARISING FROM, 
OUT OF OR IN CONNECTION WITH THE SOFTWARE OR THE USE OR OTHER DEALINGS 
IN THE SOFTWARE.
*)
IF TC.batchJobQueue.batchJobs[TC.currBatchJobIdx].state = BatchJobState.NULL THEN
	// no batchjob available
	// wait until new batchjob is loaded
ELSIF TC.batchJobQueue.batchJobs[TC.currBatchJobIdx].mode = ExecutionMode.single THEN
	SM.currW := TC.batchJobQueue.batchJobs[TC.currBatchJobIdx].workpieces[TC.batchJobQueue.batchJobs[TC.currBatchJobIdx].nextNotProcessedIdx];
	IF SM.currW.format.ejectEnabled AND NOT(SM.currW.format.furEnabled) AND NOT(SM.currW.format.sawEnabled) AND NOT(SM.currW.format.colorCheckEnabled) THEN
		// dont set SL flags because workpiece will directly be ejected HR -> VG -> EJECT
		SL.bIdx := 0;
		SL.wIdx := 0;
	ELSE
		// set SL pointers
		SL.bIdx := TC.currBatchJobIdx;
		SL.wIdx := TC.batchJobQueue.batchJobs[TC.currBatchJobIdx].nextNotProcessedIdx;
	END_IF
	TC.state := TC_State.W_LOADED;
ELSIF TC.batchJobQueue.batchJobs[TC.currBatchJobIdx].mode = ExecutionMode.multi AND (HR.state = HR_State.READY OR HR.state = HR_State.FINISHED_SINGLE_MODE OR HR.state = HR_State.SORTING) THEN
	// new w loaded in TC, load it to HR.currW
	Hr.bIdx := TC.currBatchJobIdx;
	Hr.wIdx := TC.batchJobQueue.batchJobs[TC.currBatchJobIdx].nextNotProcessedIdx;
	HR.currW := TC.batchJobQueue.batchJobs[Hr.bIdx].workpieces[Hr.wIdx];
	TC.state := TC_State.W_LOADED;
ELSIF TC.batchJobQueue.batchJobs[TC.currBatchJobIdx].mode = ExecutionMode.sorting THEN
	TC.state := TC_State.W_LOADED;
END_IF
                    
END_ACTION

ACTION start_batch_job_active:
                      (*
Copyright (c) 2019 Manuel Goester, Michael Witt, Klaus Kammerer
Institute of Databases and Information Systems, Ulm University, Germany

Permission is hereby granted, free of charge, to any person obtaining a copy 
of this software and associated documentation files (the "Software"), to deal 
in the Software without restriction, including without limitation the rights 
to use, copy, modify, merge, publish, distribute, sublicense, and/or sell 
copies of the Software, and to permit persons to whom the Software is 
furnished to do so, subject to the following conditions:

The above copyright notice and this permission notice shall be included in 
all copies or substantial portions of the Software.

THE SOFTWARE IS PROVIDED "AS IS", WITHOUT WARRANTY OF ANY KIND, EXPRESS OR 
IMPLIED, INCLUDING BUT NOT LIMITED TO THE WARRANTIES OF MERCHANTABILITY, 
FITNESS FOR A PARTICULAR PURPOSE AND NONINFRINGEMENT. IN NO EVENT SHALL THE 
AUTHORS OR COPYRIGHT HOLDERS BE LIABLE FOR ANY CLAIM, DAMAGES OR OTHER 
LIABILITY, WHETHER IN AN ACTION OF CONTRACT, TORT OR OTHERWISE, ARISING FROM, 
OUT OF OR IN CONNECTION WITH THE SOFTWARE OR THE USE OR OTHER DEALINGS 
IN THE SOFTWARE.
*)
IF started THEN
	IF NOT(fin) THEN
		IF TC.batchJobQueue.batchJobs[TC.currBatchJobIdx].state <> BatchJobState.NULL THEN
			IF TC.batchJobQueue.batchJobs[TC.currBatchJobIdx].mode = ExecutionMode.single THEN
				// start single mode
				TC.mode_active := ExecutionMode.single;
				TC.batchJobQueue.batchJobs[TC.currBatchJobIdx].state := BatchJobState.STARTED;
				fin := TRUE;
			ELSIF TC.batchJobQueue.batchJobs[TC.currBatchJobIdx].mode = ExecutionMode.multi THEN
				// start multi mode
				TC.mode_active := ExecutionMode.multi;
				TC.batchJobQueue.batchJobs[TC.currBatchJobIdx].state := BatchJobState.STARTED;
				fin := TRUE;
			ELSIF TC.batchJobQueue.batchJobs[TC.currBatchJobIdx].mode = ExecutionMode.sorting THEN
				// start sorting mode
				TC.mode_active := ExecutionMode.sorting;
				TC.batchJobQueue.batchJobs[TC.currBatchJobIdx].state := BatchJobState.STARTED;
				fin := TRUE;
			END_IF
		ELSE
			// currently no BatchJob available
			// reset HR pointers, cause they may still set
			HR.bIdx := 0;
			HR.wIdx := 0;
			HR.currW := TC.nullW;
		END_IF
	END_IF
END_IF
                    
END_ACTION

ACTION Init_active:
                      (*
Copyright (c) 2019 Manuel Goester, Michael Witt, Klaus Kammerer
Institute of Databases and Information Systems, Ulm University, Germany

Permission is hereby granted, free of charge, to any person obtaining a copy 
of this software and associated documentation files (the "Software"), to deal 
in the Software without restriction, including without limitation the rights 
to use, copy, modify, merge, publish, distribute, sublicense, and/or sell 
copies of the Software, and to permit persons to whom the Software is 
furnished to do so, subject to the following conditions:

The above copyright notice and this permission notice shall be included in 
all copies or substantial portions of the Software.

THE SOFTWARE IS PROVIDED "AS IS", WITHOUT WARRANTY OF ANY KIND, EXPRESS OR 
IMPLIED, INCLUDING BUT NOT LIMITED TO THE WARRANTIES OF MERCHANTABILITY, 
FITNESS FOR A PARTICULAR PURPOSE AND NONINFRINGEMENT. IN NO EVENT SHALL THE 
AUTHORS OR COPYRIGHT HOLDERS BE LIABLE FOR ANY CLAIM, DAMAGES OR OTHER 
LIABILITY, WHETHER IN AN ACTION OF CONTRACT, TORT OR OTHERWISE, ARISING FROM, 
OUT OF OR IN CONNECTION WITH THE SOFTWARE OR THE USE OR OTHER DEALINGS 
IN THE SOFTWARE.
*)
TC.state := TC_State.NULL;
                    
END_ACTION

ACTION Next_W_active:
                      (*
Copyright (c) 2019 Manuel Goester, Michael Witt, Klaus Kammerer
Institute of Databases and Information Systems, Ulm University, Germany

Permission is hereby granted, free of charge, to any person obtaining a copy 
of this software and associated documentation files (the "Software"), to deal 
in the Software without restriction, including without limitation the rights 
to use, copy, modify, merge, publish, distribute, sublicense, and/or sell 
copies of the Software, and to permit persons to whom the Software is 
furnished to do so, subject to the following conditions:

The above copyright notice and this permission notice shall be included in 
all copies or substantial portions of the Software.

THE SOFTWARE IS PROVIDED "AS IS", WITHOUT WARRANTY OF ANY KIND, EXPRESS OR 
IMPLIED, INCLUDING BUT NOT LIMITED TO THE WARRANTIES OF MERCHANTABILITY, 
FITNESS FOR A PARTICULAR PURPOSE AND NONINFRINGEMENT. IN NO EVENT SHALL THE 
AUTHORS OR COPYRIGHT HOLDERS BE LIABLE FOR ANY CLAIM, DAMAGES OR OTHER 
LIABILITY, WHETHER IN AN ACTION OF CONTRACT, TORT OR OTHERWISE, ARISING FROM, 
OUT OF OR IN CONNECTION WITH THE SOFTWARE OR THE USE OR OTHER DEALINGS 
IN THE SOFTWARE.
*)
// updates the current workpiece pointer to the next workpiece
IF NOT(fin) THEN
	IF NOT(TC.batchJobQueue.batchJobs[TC.currBatchJobIdx].mode = ExecutionMode.sorting) THEN
		TC.batchJobQueue.batchJobs[TC.currBatchJobIdx].nextNotProcessedIdx := TC.batchJobQueue.batchJobs[TC.currBatchJobIdx].nextNotProcessedIdx + 1;
	ELSE
		// in sorting mode always two workpieces are processed simultaniously, so increment by 2
		TC.batchJobQueue.batchJobs[TC.currBatchJobIdx].nextNotProcessedIdx := TC.batchJobQueue.batchJobs[TC.currBatchJobIdx].nextNotProcessedIdx + 2;
	END_IF
	fin := TRUE;
END_IF
                    
END_ACTION

ACTION Next_W_exit:
                      (*
Copyright (c) 2019 Manuel Goester, Michael Witt, Klaus Kammerer
Institute of Databases and Information Systems, Ulm University, Germany

Permission is hereby granted, free of charge, to any person obtaining a copy 
of this software and associated documentation files (the "Software"), to deal 
in the Software without restriction, including without limitation the rights 
to use, copy, modify, merge, publish, distribute, sublicense, and/or sell 
copies of the Software, and to permit persons to whom the Software is 
furnished to do so, subject to the following conditions:

The above copyright notice and this permission notice shall be included in 
all copies or substantial portions of the Software.

THE SOFTWARE IS PROVIDED "AS IS", WITHOUT WARRANTY OF ANY KIND, EXPRESS OR 
IMPLIED, INCLUDING BUT NOT LIMITED TO THE WARRANTIES OF MERCHANTABILITY, 
FITNESS FOR A PARTICULAR PURPOSE AND NONINFRINGEMENT. IN NO EVENT SHALL THE 
AUTHORS OR COPYRIGHT HOLDERS BE LIABLE FOR ANY CLAIM, DAMAGES OR OTHER 
LIABILITY, WHETHER IN AN ACTION OF CONTRACT, TORT OR OTHERWISE, ARISING FROM, 
OUT OF OR IN CONNECTION WITH THE SOFTWARE OR THE USE OR OTHER DEALINGS 
IN THE SOFTWARE.
*)
fin := FALSE;
                    
END_ACTION

ACTION Decide_next_W_or_BatchJob_exit:
                      (*
Copyright (c) 2019 Manuel Goester, Michael Witt, Klaus Kammerer
Institute of Databases and Information Systems, Ulm University, Germany

Permission is hereby granted, free of charge, to any person obtaining a copy 
of this software and associated documentation files (the "Software"), to deal 
in the Software without restriction, including without limitation the rights 
to use, copy, modify, merge, publish, distribute, sublicense, and/or sell 
copies of the Software, and to permit persons to whom the Software is 
furnished to do so, subject to the following conditions:

The above copyright notice and this permission notice shall be included in 
all copies or substantial portions of the Software.

THE SOFTWARE IS PROVIDED "AS IS", WITHOUT WARRANTY OF ANY KIND, EXPRESS OR 
IMPLIED, INCLUDING BUT NOT LIMITED TO THE WARRANTIES OF MERCHANTABILITY, 
FITNESS FOR A PARTICULAR PURPOSE AND NONINFRINGEMENT. IN NO EVENT SHALL THE 
AUTHORS OR COPYRIGHT HOLDERS BE LIABLE FOR ANY CLAIM, DAMAGES OR OTHER 
LIABILITY, WHETHER IN AN ACTION OF CONTRACT, TORT OR OTHERWISE, ARISING FROM, 
OUT OF OR IN CONNECTION WITH THE SOFTWARE OR THE USE OR OTHER DEALINGS 
IN THE SOFTWARE.
*)
fin := FALSE;
                    
END_ACTION

ACTION Start_Batch_Job_exit:
                      (*
Copyright (c) 2019 Manuel Goester, Michael Witt, Klaus Kammerer
Institute of Databases and Information Systems, Ulm University, Germany

Permission is hereby granted, free of charge, to any person obtaining a copy 
of this software and associated documentation files (the "Software"), to deal 
in the Software without restriction, including without limitation the rights 
to use, copy, modify, merge, publish, distribute, sublicense, and/or sell 
copies of the Software, and to permit persons to whom the Software is 
furnished to do so, subject to the following conditions:

The above copyright notice and this permission notice shall be included in 
all copies or substantial portions of the Software.

THE SOFTWARE IS PROVIDED "AS IS", WITHOUT WARRANTY OF ANY KIND, EXPRESS OR 
IMPLIED, INCLUDING BUT NOT LIMITED TO THE WARRANTIES OF MERCHANTABILITY, 
FITNESS FOR A PARTICULAR PURPOSE AND NONINFRINGEMENT. IN NO EVENT SHALL THE 
AUTHORS OR COPYRIGHT HOLDERS BE LIABLE FOR ANY CLAIM, DAMAGES OR OTHER 
LIABILITY, WHETHER IN AN ACTION OF CONTRACT, TORT OR OTHERWISE, ARISING FROM, 
OUT OF OR IN CONNECTION WITH THE SOFTWARE OR THE USE OR OTHER DEALINGS 
IN THE SOFTWARE.
*)
fin := FALSE;
                    
END_ACTION
END_PROGRAM

(* Moves HR in x and y axis Copyright (c) 2019 Manuel Goester, Michael Witt, Klaus Kammerer Institute of Databases and Information Systems, Ulm University, Germany Permission is hereby granted, free of charge, to any person obtaining a copy of this software and associated documentation files (the "Software"), to deal in the Software without restriction, including without limitation the rights to use, copy, modify, merge, publish, distribute, sublicense, and/or sell copies of the Software, and to permit persons to whom the Software is furnished to do so, subject to the following conditions: The above copyright notice and this permission notice shall be included in all copies or substantial portions of the Software. THE SOFTWARE IS PROVIDED "AS IS", WITHOUT WARRANTY OF ANY KIND, EXPRESS OR IMPLIED, INCLUDING BUT NOT LIMITED TO THE WARRANTIES OF MERCHANTABILITY, FITNESS FOR A PARTICULAR PURPOSE AND NONINFRINGEMENT. IN NO EVENT SHALL THE AUTHORS OR COPYRIGHT HOLDERS BE LIABLE FOR ANY CLAIM, DAMAGES OR OTHER LIABILITY, WHETHER IN AN ACTION OF CONTRACT, TORT OR OTHERWISE, ARISING FROM, OUT OF OR IN CONNECTION WITH THE SOFTWARE OR THE USE OR OTHER DEALINGS IN THE SOFTWARE. *)
FUNCTION_BLOCK HR_MOVE
  VAR_INPUT
    x : INT;  (* distance HR will go right (negative value) or left (positive value) *)
    y : INT;  (* distance HR will go up (negative value) or down (positive value) *)
  END_VAR
  VAR
    xFin : BOOL := FALSE;  (* finish flags *)
    yFin : BOOL := FALSE;
    fin : BOOL := FALSE;
    xAlreadyCounted : BOOL := FALSE;  (* true, if an impulse coming from the motor has been already counted *)
    yAlreadyCounted : BOOL := FALSE;
    cX : INT := 0;  (* counters for x and y axis *)
    cY : INT := 0;
  END_VAR

                  fin := FALSE;

// X AXIS
IF x < 0 THEN
	// drive right
	IF cX = x THEN
		// if counter reached demanded position, we're done
		HR.mHorizontalRight := FALSE;
		HR.mHorizontalLeft := FALSE;
		xFin := TRUE;
	ELSE
		xFin := FALSE;
		IF cX > x THEN
			HR.mHorizontalRight := TRUE;
			IF HR.encHorizontal AND NOT(xAlreadyCounted) THEN
				// update local counter
				cX := cX - 1;
				// update global counter
				HR.cX := HR.cX - 1;
				xAlreadyCounted := TRUE;
			ELSIF NOT(HR.encHorizontal) THEN
				xAlreadyCounted := FALSE;
			END_IF
		END_IF
	END_IF
ELSE
	// x >= 0
	// drive left
	IF cX = x THEN
		// if counter reached demanded position, we're done
		HR.mHorizontalRight := FALSE;
		HR.mHorizontalLeft := FALSE;
		xFin := TRUE;
	ELSE
		xFin := FALSE;
		IF cX < x THEN
			HR.mHorizontalLeft := TRUE;
			IF HR.encHorizontal AND NOT(xAlreadyCounted) THEN
				// update local counter
				cX := cX + 1;
				// update global counter
				HR.cX := HR.cX + 1;
				xAlreadyCounted := TRUE;
			ELSIF NOT(HR.encHorizontal) THEN
				xAlreadyCounted := FALSE;
			END_IF
		END_IF
	END_IF
END_IF

// Y AXIS
IF y < 0 THEN
	// drive up
	IF cY = y THEN
		// if counter reached demanded position, we're done
		HR.mVerticalUp := FALSE;
		HR.mVerticalDown := FALSE;
		yFin := TRUE;
	ELSE
		yFin := FALSE;
		IF cY > y THEN
			HR.mVerticalUp := TRUE;
			IF HR.encVertical AND NOT(yAlreadyCounted) THEN
				// update local counter
				cY := cY - 1;
				// update global counter
				HR.cY := HR.cY - 1;
				yAlreadyCounted := TRUE;
			ELSIF NOT(HR.encVertical) THEN
				yAlreadyCounted := FALSE;
			END_IF
		END_IF
	END_IF
ELSE
	// y >= 0
	// drive down
	IF cY = y THEN
		// if counter reached demanded position, we're done
		HR.mVerticalDown := FALSE;
		HR.mVerticalUp := FALSE;
	yFin := TRUE;
	ELSE
		yFin := FALSE;
		IF cY < y THEN
			HR.mVerticalDown := TRUE;
			IF HR.encVertical AND NOT(yAlreadyCounted) THEN
				// update local counter
				cY := cY + 1;
				// update global counter
				HR.cY := HR.cY + 1;
				yAlreadyCounted := TRUE;
			ELSIF NOT(HR.encVertical) THEN
				yAlreadyCounted := FALSE;
			END_IF
		END_IF
	END_IF
END_IF

// if x and y axis are finsihed, we're done
IF xFin AND yFin THEN
	// reset local counters
	cX := 0;
	cY := 0;
	xFin := FALSE;
	yFin := FALSE;
	fin := TRUE;
	RETURN;
END_IF
                
END_FUNCTION_BLOCK

PROGRAM FUR_MULTI_MODE
  VAR
    fur_burn : FUR_BURN;
    timer : TON;
    finBurner : BOOL := FALSE;
    stepSuccer : INT := 1;
    stepSaw : INT := 1;
    fin : BOOL;
    counter : INT;
  END_VAR

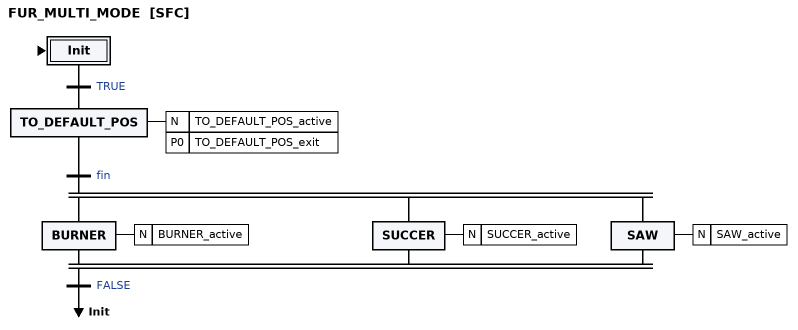
INITIAL_STEP Init:
END_STEP
TRANSITION FROM Init TO TO_DEFAULT_POS
  := TRUE;
END_TRANSITION
STEP TO_DEFAULT_POS:
  TO_DEFAULT_POS_active(N);
  TO_DEFAULT_POS_exit(P0);
END_STEP
TRANSITION FROM TO_DEFAULT_POS TO (BURNER, SUCCER, SAW)
  := fin;
END_TRANSITION
STEP BURNER:
  BURNER_active(N);
END_STEP
TRANSITION FROM (BURNER, SUCCER, SAW) TO Init
  := FALSE;
END_TRANSITION
STEP SUCCER:
  SUCCER_active(N);
END_STEP
STEP SAW:
  SAW_active(N);
END_STEP

ACTION BURNER_active:
                      (*
Copyright (c) 2019 Manuel Goester, Michael Witt, Klaus Kammerer
Institute of Databases and Information Systems, Ulm University, Germany

Permission is hereby granted, free of charge, to any person obtaining a copy 
of this software and associated documentation files (the "Software"), to deal 
in the Software without restriction, including without limitation the rights 
to use, copy, modify, merge, publish, distribute, sublicense, and/or sell 
copies of the Software, and to permit persons to whom the Software is 
furnished to do so, subject to the following conditions:

The above copyright notice and this permission notice shall be included in 
all copies or substantial portions of the Software.

THE SOFTWARE IS PROVIDED "AS IS", WITHOUT WARRANTY OF ANY KIND, EXPRESS OR 
IMPLIED, INCLUDING BUT NOT LIMITED TO THE WARRANTIES OF MERCHANTABILITY, 
FITNESS FOR A PARTICULAR PURPOSE AND NONINFRINGEMENT. IN NO EVENT SHALL THE 
AUTHORS OR COPYRIGHT HOLDERS BE LIABLE FOR ANY CLAIM, DAMAGES OR OTHER 
LIABILITY, WHETHER IN AN ACTION OF CONTRACT, TORT OR OTHERWISE, ARISING FROM, 
OUT OF OR IN CONNECTION WITH THE SOFTWARE OR THE USE OR OTHER DEALINGS 
IN THE SOFTWARE.
*)
IF FUR.currWBurner.state <> W_State.NULL THEN
	// fur burner got an w
	IF FUR.currWBurner.format.furEnabled AND NOT(finBurner) THEN
		// burn
		fur_burn(w := FUR.currWBurner);
		finBurner := fur_burn.fin;
	ELSE
		IF FUR.currWSuccer.state = W_State.NULL THEN
			// bend pointers of fur succer to current workpiece
			counter := counter + 1;
			
			FUR.bIdxSuccer := FUR.bIdxBurner;
			FUR.wIdxSuccer := FUR.wIdxBurner;
			FUR.currWSuccer := TC.batchJobQueue.batchJobs[FUR.bIdxSuccer].workpieces[FUR.wIdxSuccer];
			// reset own pointers
			FUR.bIdxBurner := 0;
			FUR.wIdxBurner := 0;
			FUR.currWBurner := TC.nullW;
			finBurner := FALSE;
		END_IF
	END_IF
END_IF
                    
END_ACTION

ACTION SUCCER_active:
                      (*
Copyright (c) 2019 Manuel Goester, Michael Witt, Klaus Kammerer
Institute of Databases and Information Systems, Ulm University, Germany

